KUKA KRL program: MyProgram_111().src

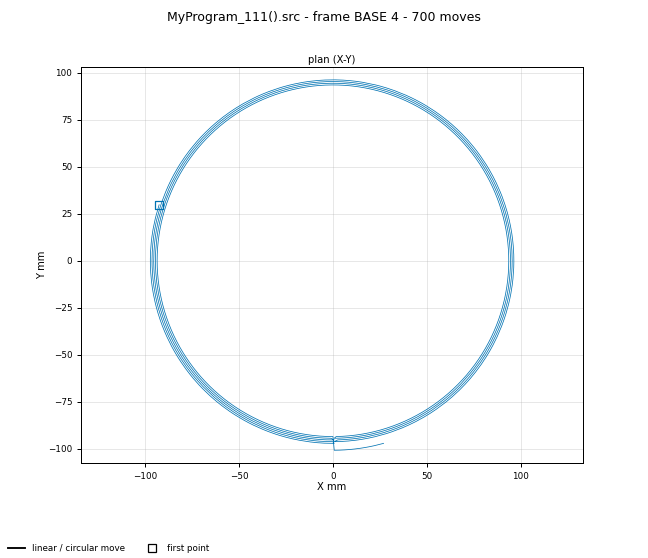
[picture p0: tool path of MyProgram_111().src in frame BASE 4, 700 of 700 moves have a stored position in this frame; points joined in program order, loops and branches not executed]
&ACCESS RVP
&REL 1
&PARAM TEMPLATE = C:\KRC\Roboter\Template\vorgabe
&PARAM EDITMASK = *
DEF MyProgram_111()
; ---- Setting reference (Base) ----
$BASE = BASE_DATA[4]

; --------------------------
; ---- Setting tool (TCP) ----
$TOOL = TOOL_DATA[3]
; --------------------------

$VEL.CP = VEL_APROX_PRINT
Startdeposition()
$VEL.CP = VEL_PRINT
LIN {X -92.4915,Y 29.7946,Z 97,A 157.868,B 24.9225,C -2.0326,E1 24.8471,E2 287.401} C_DIS
LIN {X -94.4382,Y 22.8874,Z 97,A 162.0208,B 24.9237,C -2.0166,E1 24.844,E2 283.2622} C_DIS
LIN {X -95.7031,Y 16.8359,Z 97,A 165.9283,B 24.924,C -2.0135,E1 24.8419,E2 279.3391} C_DIS
LIN {X -96.2599,Y 13.2878,Z 97,A 167.8285,B 24.925,C -1.9996,E1 24.8411,E2 277.4607} C_DIS
LIN {X -96.6738,Y 9.8311,Z 97,A 170.0082,B 24.9252,C -1.9971,E1 24.8405,E2 275.2738} C_DIS
LIN {X -97.0459,Y 4.9634,Z 97,A 172.6353,B 24.9265,C -1.9797,E1 24.84,E2 272.6726} C_DIS
LIN {X -97.1667,Y 1.1606,Z 97,A 174.9618,B 24.9269,C -1.9751,E1 24.8398,E2 270.3429} C_DIS
LIN {X -97.1555,Y -1.7889,Z 97,A 176.8668,B 24.9269,C -1.975,E1 24.8398,E2 268.4268} C_DIS
LIN {X -96.9581,Y -6.4444,Z 97,A 179.9808,B 24.9266,C -1.9782,E1 24.8403,E2 265.2864} C_DIS
LIN {X -96.5322,Y -11.1337,Z 97,A -177.5959,B 24.9281,C -1.9578,E1 24.841,E2 262.8972} C_DIS
LIN {X -96.1039,Y -14.3757,Z 97,A -175.1891,B 24.9274,C -1.9674,E1 24.842,E2 260.4532} C_DIS
LIN {X -95.5709,Y -17.5708,Z 97,A -174.0896,B 24.9298,C -1.9349,E1 24.8425,E2 259.4247} C_DIS
LIN {X -94.6671,Y -21.921,Z 97,A -171.138,B 24.9296,C -1.9376,E1 24.8442,E2 256.4493} C_DIS
LIN {X -94.0208,Y -24.5484,Z 97,A -168.9937,B 24.9287,C -1.9508,E1 24.8458,E2 254.261} C_DIS
LIN {X -93.1291,Y -27.7365,Z 97,A -167.1259,B 24.9293,C -1.9421,E1 24.8472,E2 252.4031} C_DIS
LIN {X -91.8935,Y -31.5962,Z 97,A -165.2192,B 24.931,C -1.919,E1 24.8489,E2 250.5406} C_DIS
LIN {X -90.915,Y -34.3054,Z 97,A -163.416,B 24.931,C -1.9175,E1 24.8506,E2 248.7308} C_DIS
LIN {X -89.6794,Y -37.418,Z 97,A -161.4125,B 24.9314,C -1.9127,E1 24.8527,E2 246.7275} C_DIS
LIN {X -88.3292,Y -40.505,Z 97,A -158.9881,B 24.9308,C -1.9216,E1 24.8556,E2 244.2687} C_DIS
LIN {X -85.934,Y -45.3624,Z 97,A -155.9633,B 24.9318,C -1.9072,E1 24.8594,E2 241.262} C_DIS
LIN {X -84.4252,Y -48.1133,Z 97,A -154.2857,B 24.9326,C -1.8964,E1 24.8617,E2 239.6013} C_DIS
LIN {X -82.6777,Y -51.0591,Z 97,A -152.4701,B 24.9334,C -1.8843,E1 24.8642,E2 237.8053} C_DIS
LIN {X -81.1737,Y -53.4156,Z 97,A -150.6577,B 24.9334,C -1.8856,E1 24.867,E2 235.9808} C_DIS
LIN {X -78.2895,Y -57.5602,Z 97,A -147.9461,B 24.9345,C -1.8692,E1 24.8714,E2 233.2948} C_DIS
LIN {X -76.0614,Y -60.4742,Z 97,A -145.6413,B 24.9345,C -1.8687,E1 24.8753,E2 230.9802} C_DIS
LIN {X -74.3345,Y -62.5867,Z 97,A -143.0069,B 24.9323,C -1.8998,E1 24.8802,E2 228.2597} C_DIS
LIN {X -71.1942,Y -66.1371,Z 97,A -141.1694,B 24.9351,C -1.8609,E1 24.8835,E2 226.5067} C_DIS
LIN {X -69.3992,Y -68.0168,Z 97,A -138.452,B 24.9325,C -1.8982,E1 24.889,E2 223.6888} C_DIS
LIN {X -65.4486,Y -71.8261,Z 97,A -136.4982,B 24.936,C -1.8476,E1 24.8928,E2 221.8475} C_DIS
LIN {X -61.836,Y -74.9588,Z 97,A -133.6287,B 24.9363,C -1.8439,E1 24.8989,E2 218.9758} C_DIS
LIN {X -59.0106,Y -77.2029,Z 97,A -131.1944,B 24.9358,C -1.8506,E1 24.9043,E2 216.5166} C_DIS
LIN {X -55.0989,Y -80.0414,Z 97,A -127.9514,B 24.9352,C -1.8594,E1 24.9117,E2 213.2414} C_DIS
LIN {X -52.3049,Y -81.8941,Z 97,A -126.3944,B 24.9364,C -1.8418,E1 24.9153,E2 211.7214} C_DIS
LIN {X -47.6565,Y -84.6838,Z 97,A -123.5051,B 24.9375,C -1.8265,E1 24.9222,E2 208.8597} C_DIS
LIN {X -44.9402,Y -86.1564,Z 97,A -121.5459,B 24.9373,C -1.8289,E1 24.927,E2 206.8894} C_DIS
LIN {X -42.2462,Y -87.5082,Z 97,A -119.4558,B 24.9367,C -1.8377,E1 24.9323,E2 204.7729} C_DIS
LIN {X -37.2841,Y -89.7359,Z 97,A -116.4957,B 24.9375,C -1.8255,E1 24.9399,E2 201.8348} C_DIS
LIN {X -34.0837,Y -90.9986,Z 97,A -114.3639,B 24.9375,C -1.8272,E1 24.9454,E2 199.6942} C_DIS
LIN {X -30.4442,Y -92.2814,Z 97,A -112.2394,B 24.9379,C -1.82,E1 24.951,E2 197.583} C_DIS
LIN {X -28.0314,Y -93.0419,Z 97,A -110.5722,B 24.9376,C -1.8251,E1 24.9555,E2 195.9006} C_DIS
LIN {X -24.7478,Y -93.9695,Z 97,A -108.1059,B 24.9365,C -1.8402,E1 24.9623,E2 193.3949} C_DIS
LIN {X -21.4833,Y -94.7682,Z 97,A -106.8785,B 24.9384,C -1.8121,E1 24.9654,E2 192.2324} C_DIS
LIN {X -17.7571,Y -95.5374,Z 97,A -104.2589,B 24.9376,C -1.8247,E1 24.9727,E2 189.58} C_DIS
LIN {X -12.0154,Y -96.4274,Z 97,A -100.8841,B 24.9378,C -1.822,E1 24.982,E2 186.2087} C_DIS
LIN {X -8.4428,Y -96.8057,Z 97,A -98.2149,B 24.9364,C -1.842,E1 24.9896,E2 183.4909} C_DIS
LIN {X -4.6237,Y -97.0629,Z 97,A -96.7543,B 24.9384,C -1.813,E1 24.9935,E2 182.0985} C_DIS
LIN {X 0.694,Y -97.1695,Z 97,A -93.9172,B 24.9391,C -1.8027,E1 25.0013,E2 179.2858} C_DIS
Enddeposition()
LIN {X 0.694,Y -97.1695,Z 97,A -93.9172,B 24.9391,C -1.8027,E1 25.0013,E2 179.2858} C_DIS
Startdeposition()
$VEL.CP = VEL_PRINT
LIN {X -0.1063,Y -96.2686,Z 97,A -95.3472,B 24.9403,C -1.7844,E1 24.9972,E2 180.7591} C_DIS
LIN {X -3.6596,Y -96.1991,Z 97,A -96.7459,B 24.9386,C -1.8095,E1 24.9935,E2 182.0986} C_DIS
LIN {X -7.1701,Y -96.0013,Z 97,A -99.0523,B 24.9391,C -1.8018,E1 24.987,E2 184.4239} C_DIS
LIN {X -10.3776,Y -95.7072,Z 97,A -101.037,B 24.9393,C -1.7996,E1 24.9814,E2 186.4149} C_DIS
LIN {X -16.5386,Y -94.8376,Z 97,A -104.7525,B 24.9393,C -1.8001,E1 24.9712,E2 190.1325} C_DIS
LIN {X -20.308,Y -94.1013,Z 97,A -106.7067,B 24.9384,C -1.8127,E1 24.9659,E2 192.0591} C_DIS
LIN {X -22.8168,Y -93.5244,Z 97,A -108.7921,B 24.9397,C -1.7943,E1 24.9601,E2 194.1911} C_DIS
LIN {X -27.203,Y -92.3442,Z 97,A -111.1051,B 24.9386,C -1.8095,E1 24.954,E2 196.4716} C_DIS
LIN {X -30.6307,Y -91.2645,Z 97,A -113.1926,B 24.9384,C -1.8129,E1 24.9484,E2 198.5547} C_DIS
LIN {X -33.6837,Y -90.1833,Z 97,A -115.2946,B 24.9387,C -1.8086,E1 24.9429,E2 200.6712} C_DIS
LIN {X -36.8901,Y -88.9204,Z 97,A -117.1546,B 24.9381,C -1.8172,E1 24.9381,E2 202.5149} C_DIS
LIN {X -42.0764,Y -86.5863,Z 97,A -120.7767,B 24.9384,C -1.8129,E1 24.9289,E2 206.1561} C_DIS
LIN {X -44.7962,Y -85.2099,Z 97,A -122.6012,B 24.9383,C -1.8149,E1 24.9243,E2 207.9809} C_DIS
LIN {X -47.0298,Y -83.9978,Z 97,A -124.2047,B 24.9383,C -1.8139,E1 24.9204,E2 209.5914} C_DIS
LIN {X -50.4531,Y -81.989,Z 97,A -126.5088,B 24.938,C -1.8192,E1 24.9149,E2 211.8897} C_DIS
LIN {X -52.931,Y -80.4098,Z 97,A -128.9407,B 24.9393,C -1.7993,E1 24.9091,E2 214.3772} C_DIS
LIN {X -56.6092,Y -77.8648,Z 97,A -130.8407,B 24.9373,C -1.829,E1 24.905,E2 216.213} C_DIS
LIN {X -58.4653,Y -76.4812,Z 97,A -132.5565,B 24.9379,C -1.8202,E1 24.9011,E2 217.9559} C_DIS
LIN {X -62.9436,Y -72.8408,Z 97,A -135.7325,B 24.9369,C -1.8353,E1 24.8943,E2 221.1083} C_DIS
LIN {X -69.1499,Y -66.9759,Z 97,A -140.5168,B 24.9355,C -1.8556,E1 24.8847,E2 225.8638} C_DIS
LIN {X -73.3934,Y -62.2966,Z 97,A -144.6286,B 24.9357,C -1.8524,E1 24.877,E2 230.0016} C_DIS
LIN {X -75.3487,Y -59.9173,Z 97,A -146.6761,B 24.9359,C -1.8498,E1 24.8734,E2 232.0651} C_DIS
LIN {X -77.8768,Y -56.5928,Z 97,A -149.3083,B 24.9358,C -1.8511,E1 24.869,E2 234.7068} C_DIS
LIN {X -80.6335,Y -52.5917,Z 97,A -151.6927,B 24.9341,C -1.8749,E1 24.8654,E2 237.0464} C_DIS
LIN {X -81.8943,Y -50.6061,Z 97,A -153.2387,B 24.9341,C -1.8738,E1 24.8631,E2 238.6028} C_DIS
LIN {X -83.5244,Y -47.8655,Z 97,A -155.0065,B 24.9335,C -1.8831,E1 24.8606,E2 240.3577} C_DIS
LIN {X -85.7783,Y -43.6981,Z 97,A -157.9857,B 24.9333,C -1.8857,E1 24.8567,E2 243.3466} C_DIS
LIN {X -87.5768,Y -39.9744,Z 97,A -160.4617,B 24.9329,C -1.8921,E1 24.8537,E2 245.8207} C_DIS
LIN {X -88.8678,Y -37.0149,Z 97,A -162.449,B 24.9326,C -1.8955,E1 24.8516,E2 247.8109} C_DIS
LIN {X -90.1653,Y -33.7313,Z 97,A -164.534,B 24.9322,C -1.9022,E1 24.8495,E2 249.8917} C_DIS
LIN {X -91.1712,Y -30.9074,Z 97,A -167.3212,B 24.934,C -1.8758,E1 24.847,E2 252.7577} C_DIS
LIN {X -92.7753,Y -25.7,Z 97,A -169.5931,B 24.9312,C -1.9162,E1 24.8453,E2 254.9465} C_DIS
LIN {X -93.6014,Y -22.5015,Z 97,A -172.0952,B 24.9319,C -1.9053,E1 24.8436,E2 257.4892} C_DIS
LIN {X -94.3933,Y -18.9045,Z 97,A -173.5687,B 24.9298,C -1.9348,E1 24.8428,E2 258.9009} C_DIS
LIN {X -95.3216,Y -13.462,Z 97,A -176.997,B 24.9294,C -1.9405,E1 24.8412,E2 262.3358} C_DIS
LIN {X -95.7625,Y -9.8494,Z 97,A -179.7199,B 24.9302,C -1.9299,E1 24.8404,E2 265.1006} C_DIS
LIN {X -96.0521,Y -6.4361,Z 97,A 178.1629,B 24.9299,C -1.9339,E1 24.84,E2 267.2209} C_DIS
LIN {X -96.2279,Y -2.7676,Z 97,A 176.4444,B 24.9283,C -1.9556,E1 24.8398,E2 268.898} C_DIS
LIN {X -96.2681,Y 0.3084,Z 97,A 173.9579,B 24.9294,C -1.9409,E1 24.8398,E2 271.4346} C_DIS
LIN {X -96.1614,Y 4.5356,Z 97,A 172.4406,B 24.9265,C -1.9804,E1 24.84,E2 272.8668} C_DIS
LIN {X -95.8516,Y 8.9387,Z 97,A 169.4889,B 24.9266,C -1.9785,E1 24.8406,E2 275.8406} C_DIS
LIN {X -95.4419,Y 12.5827,Z 97,A 167.4434,B 24.9258,C -1.9899,E1 24.8413,E2 277.8713} C_DIS
LIN {X -94.8189,Y 16.6424,Z 97,A 164.3977,B 24.9266,C -1.9788,E1 24.8427,E2 280.9615} C_DIS
LIN {X -94.2033,Y 19.8342,Z 97,A 162.8144,B 24.9253,C -1.996,E1 24.8436,E2 282.5132} C_DIS
LIN {X -93.6552,Y 22.2809,Z 97,A 160.0692,B 24.9279,C -1.9616,E1 24.8455,E2 285.3564} C_DIS
LIN {X -91.9819,Y 28.4036,Z 97,A 157.5986,B 24.9239,C -2.0142,E1 24.8473,E2 287.7158} C_DIS
LIN {X -90.9839,Y 31.4572,Z 97,A 154.5779,B 24.9261,C -1.9854,E1 24.8502,E2 290.8223} C_DIS
LIN {X -89.0472,Y 36.5773,Z 97,A 151.982,B 24.9238,C -2.0161,E1 24.8528,E2 293.3597} C_DIS
LIN {X -87.6404,Y 39.8331,Z 97,A 149.8079,B 24.9235,C -2.0204,E1 24.8553,E2 295.5354} C_DIS
LIN {X -86.2622,Y 42.7349,Z 97,A 147.841,B 24.9232,C -2.0243,E1 24.8578,E2 297.5034} C_DIS
LIN {X -84.6982,Y 45.7566,Z 97,A 146.652,B 24.9207,C -2.0568,E1 24.8592,E2 298.6213} C_DIS
LIN {X -82.7301,Y 49.2264,Z 97,A 144.0967,B 24.9206,C -2.0578,E1 24.8628,E2 301.1876} C_DIS
LIN {X -81.391,Y 51.41,Z 97,A 142.0984,B 24.9214,C -2.047,E1 24.8658,E2 303.2218} C_DIS
LIN {X -78.721,Y 55.4119,Z 97,A 139.1346,B 24.9211,C -2.0517,E1 24.8705,E2 306.1889} C_DIS
LIN {X -76.305,Y 58.6939,Z 97,A 136.7507,B 24.9205,C -2.0596,E1 24.8745,E2 308.5656} C_DIS
LIN {X -72.7774,Y 63.0162,Z 97,A 133.1858,B 24.9204,C -2.0604,E1 24.8809,E2 312.145} C_DIS
LIN {X -70.4253,Y 65.6345,Z 97,A 131.55,B 24.9188,C -2.0803,E1 24.884,E2 313.7405} C_DIS
LIN {X -67.6647,Y 68.4757,Z 97,A 128.6745,B 24.9197,C -2.0694,E1 24.8897,E2 316.6542} C_DIS
LIN {X -65.0275,Y 70.9849,Z 97,A 126.5163,B 24.9193,C -2.0746,E1 24.8941,E2 318.8085} C_DIS
LIN {X -62.3518,Y 73.3464,Z 97,A 124.8919,B 24.9176,C -2.0955,E1 24.8975,E2 320.3895} C_DIS
LIN {X -58.4338,Y 76.5045,Z 97,A 121.6806,B 24.9176,C -2.0949,E1 24.9046,E2 323.6142} C_DIS
LIN {X -54.9913,Y 79.0151,Z 97,A 119.1069,B 24.9174,C -2.0988,E1 24.9104,E2 326.1874} C_DIS
LIN {X -51.533,Y 81.3147,Z 97,A 116.1285,B 24.9183,C -2.087,E1 24.9175,E2 329.2035} C_DIS
LIN {X -47.8726,Y 83.5204,Z 97,A 113.9285,B 24.9171,C -2.1027,E1 24.9228,E2 331.3726} C_DIS
LIN {X -41.8924,Y 86.6747,Z 97,A 110.3041,B 24.9155,C -2.1225,E1 24.9317,E2 334.9598} C_DIS
LIN {X -39.8287,Y 87.6424,Z 97,A 108.8219,B 24.9157,C -2.1204,E1 24.9355,E2 336.4507} C_DIS
LIN {X -37.2678,Y 88.7612,Z 97,A 107.175,B 24.9154,C -2.1233,E1 24.9397,E2 338.0944} C_DIS
LIN {X -33.9421,Y 90.0855,Z 97,A 105.1375,B 24.915,C -2.1293,E1 24.945,E2 340.1221} C_DIS
LIN {X -28.5804,Y 91.9271,Z 97,A 102.0567,B 24.9139,C -2.1432,E1 24.9531,E2 343.1756} C_DIS
LIN {X -26.6002,Y 92.5198,Z 97,A 99.971,B 24.916,C -2.1158,E1 24.9588,E2 345.3298} C_DIS
LIN {X -23.1497,Y 93.4432,Z 97,A 98.3572,B 24.9145,C -2.135,E1 24.9631,E2 346.9002} C_DIS
LIN {X -20.474,Y 94.0651,Z 97,A 96.4503,B 24.9151,C -2.1273,E1 24.9683,E2 348.8278} C_DIS
LIN {X -15.9853,Y 94.9311,Z 97,A 94.0207,B 24.9142,C -2.1393,E1 24.9749,E2 351.2315} C_DIS
LIN {X -12.802,Y 95.4134,Z 97,A 92.0226,B 24.9142,C -2.1377,E1 24.9805,E2 353.235} C_DIS
LIN {X -7.6508,Y 95.963,Z 97,A 89.0303,B 24.9139,C -2.1424,E1 24.9888,E2 356.2177} C_DIS
LIN {X -4.163,Y 96.1774,Z 97,A 86.9285,B 24.9139,C -2.1424,E1 24.9946,E2 358.3201} C_DIS
LIN {X 1.1849,Y 96.262,Z 97,A 83.4209,B 24.9148,C -2.1319,E1 25.0045,E2 361.8527} C_DIS
LIN {X 5.3529,Y 96.1185,Z 97,A 81.2928,B 24.9138,C -2.1443,E1 25.0103,E2 363.9506} C_DIS
LIN {X 8.6175,Y 95.8813,Z 97,A 79.3012,B 24.9138,C -2.1426,E1 25.0159,E2 365.9451} C_DIS
LIN {X 12.1982,Y 95.4917,Z 97,A 77.1548,B 24.9139,C -2.1422,E1 25.0218,E2 368.091} C_DIS
LIN {X 15.6937,Y 94.9798,Z 97,A 74.8864,B 24.9145,C -2.1357,E1 25.0281,E2 370.3725} C_DIS
LIN {X 22.781,Y 93.5332,Z 97,A 70.7418,B 24.9142,C -2.1393,E1 25.0394,E2 374.5033} C_DIS
LIN {X 25.0573,Y 92.9492,Z 97,A 69.1352,B 24.9148,C -2.1311,E1 25.0438,E2 376.1269} C_DIS
LIN {X 28.7594,Y 91.8716,Z 97,A 66.8778,B 24.9148,C -2.1307,E1 25.0498,E2 378.3813} C_DIS
LIN {X 32.8246,Y 90.4986,Z 97,A 64.5081,B 24.9145,C -2.135,E1 25.056,E2 380.736} C_DIS
LIN {X 38.8687,Y 88.0729,Z 97,A 60.6771,B 24.9147,C -2.1326,E1 25.0659,E2 384.5638} C_DIS
LIN {X 41.7242,Y 86.7555,Z 97,A 58.6642,B 24.9153,C -2.1253,E1 25.071,E2 386.5889} C_DIS
LIN {X 44.0379,Y 85.6046,Z 97,A 56.6873,B 24.9167,C -2.1074,E1 25.076,E2 388.6025} C_DIS
LIN {X 47.3152,Y 83.8385,Z 97,A 54.9623,B 24.9155,C -2.1221,E1 25.0801,E2 390.2878} C_DIS
LIN {X 49.6095,Y 82.5017,Z 97,A 52.5123,B 24.9182,C -2.0883,E1 25.0862,E2 392.8101} C_DIS
LIN {X 53.8888,Y 79.7711,Z 97,A 50.4443,B 24.9159,C -2.118,E1 25.0908,E2 394.801} C_DIS
LIN {X 56.8975,Y 77.6537,Z 97,A 48.1904,B 24.9164,C -2.1119,E1 25.0959,E2 397.0615} C_DIS
LIN {X 59.7862,Y 75.4523,Z 97,A 46.0467,B 24.9166,C -2.1086,E1 25.1006,E2 399.205} C_DIS
LIN {X 63.1591,Y 72.6526,Z 97,A 42.8742,B 24.9186,C -2.0829,E1 25.1075,E2 402.4259} C_DIS
LIN {X 66.1256,Y 69.9635,Z 97,A 41.057,B 24.9174,C -2.0988,E1 25.1111,E2 404.198} C_DIS
LIN {X 68.6689,Y 67.4691,Z 97,A 38.8708,B 24.9179,C -2.0918,E1 25.1154,E2 406.3914} C_DIS
LIN {X 71.4686,Y 64.4966,Z 97,A 36.5932,B 24.9179,C -2.0921,E1 25.1197,E2 408.6584} C_DIS
LIN {X 73.095,Y 62.6468,Z 97,A 35.2236,B 24.9179,C -2.0924,E1 25.1222,E2 410.0212} C_DIS
LIN {X 75.1292,Y 60.1941,Z 97,A 33.3527,B 24.9182,C -2.0888,E1 25.1255,E2 411.8918} C_DIS
LIN {X 76.6102,Y 58.2967,Z 97,A 31.8354,B 24.9187,C -2.0822,E1 25.1281,E2 413.4176} C_DIS
LIN {X 78.5024,Y 55.7212,Z 97,A 30.0024,B 24.9189,C -2.0801,E1 25.1311,E2 415.2468} C_DIS
LIN {X 81.6082,Y 51.0639,Z 97,A 26.652,B 24.9196,C -2.0708,E1 25.1362,E2 418.6024} C_DIS
LIN {X 83.1374,Y 48.5373,Z 97,A 24.1439,B 24.9221,C -2.0378,E1 25.1399,E2 421.1753} C_DIS
LIN {X 85.2358,Y 44.7471,Z 97,A 22.2783,B 24.9206,C -2.0576,E1 25.1422,E2 422.9844} C_DIS
LIN {X 86.8297,Y 41.5699,Z 97,A 20.4727,B 24.9202,C -2.0635,E1 25.1444,E2 424.7665} C_DIS
LIN {X 89.0364,Y 36.6069,Z 97,A 17.0287,B 24.9215,C -2.0461,E1 25.1483,E2 428.2326} C_DIS
LIN {X 89.9521,Y 34.2941,Z 97,A 14.7796,B 24.924,C -2.0127,E1 25.1506,E2 430.5481} C_DIS
LIN {X 91.4513,Y 30.0714,Z 97,A 12.1056,B 24.9247,C -2.0044,E1 25.1529,E2 433.2265} C_DIS
LIN {X 92.7719,Y 25.712,Z 97,A 10.1116,B 24.9232,C -2.0234,E1 25.1544,E2 435.1643} C_DIS
LIN {X 93.8162,Y 21.5858,Z 97,A 7.6077,B 24.9237,C -2.0167,E1 25.1561,E2 437.6694} C_DIS
LIN {X 94.5734,Y 17.9821,Z 97,A 5.4465,B 24.9242,C -2.0111,E1 25.1573,E2 439.8314} C_DIS
LIN {X 95.1599,Y 14.5614,Z 97,A 3.4483,B 24.9245,C -2.0072,E1 25.1581,E2 441.827} C_DIS
LIN {X 95.6181,Y 11.1625,Z 97,A 1.4693,B 24.9248,C -2.0031,E1 25.1588,E2 443.8039} C_DIS
LIN {X 95.947,Y 7.8507,Z 97,A -0.5562,B 24.9254,C -1.9951,E1 25.1594,E2 445.8364} C_DIS
LIN {X 96.2103,Y 3.3404,Z 97,A -3.7404,B 24.9274,C -1.9675,E1 25.1598,E2 449.0668} C_DIS
LIN {X 96.2683,Y -0.2759,Z 97,A -5.409,B 24.9266,C -1.9791,E1 25.1598,E2 450.698} C_DIS
LIN {X 96.1914,Y -3.8381,Z 97,A -7.1655,B 24.926,C -1.9863,E1 25.1596,E2 452.427} C_DIS
LIN {X 95.7875,Y -9.6102,Z 97,A -10.892,B 24.9277,C -1.9643,E1 25.1589,E2 456.1835} C_DIS
LIN {X 95.3861,Y -13.0079,Z 97,A -12.9595,B 24.9282,C -1.9565,E1 25.1581,E2 458.2571} C_DIS
LIN {X 94.6398,Y -17.6367,Z 97,A -15.7128,B 24.9288,C -1.949,E1 25.1568,E2 461.012} C_DIS
LIN {X 94.1134,Y -20.2525,Z 97,A -17.2967,B 24.9291,C -1.9441,E1 25.1559,E2 462.5982} C_DIS
LIN {X 93.4103,Y -23.2847,Z 97,A -19.3832,B 24.9302,C -1.9292,E1 25.1545,E2 464.7078} C_DIS
LIN {X 92.0627,Y -28.143,Z 97,A -22.0736,B 24.93,C -1.9317,E1 25.1524,E2 467.377} C_DIS
LIN {X 91.0382,Y -31.3019,Z 97,A -24.0007,B 24.9304,C -1.9274,E1 25.1507,E2 469.3033} C_DIS
LIN {X 89.7528,Y -34.8143,Z 97,A -26.5939,B 24.9319,C -1.9064,E1 25.1481,E2 471.9314} C_DIS
LIN {X 87.3524,Y -40.4601,Z 97,A -29.9301,B 24.9318,C -1.9074,E1 25.1444,E2 475.247} C_DIS
LIN {X 85.121,Y -44.965,Z 97,A -33.3271,B 24.9335,C -1.8831,E1 25.14,E2 478.6835} C_DIS
LIN {X 83.4643,Y -47.9701,Z 97,A -34.9806,B 24.9329,C -1.892,E1 25.1378,E2 480.3074} C_DIS
LIN {X 81.504,Y -51.2308,Z 97,A -36.8015,B 24.9321,C -1.9025,E1 25.1352,E2 482.0942} C_DIS
LIN {X 78.9338,Y -55.1082,Z 97,A -39.7281,B 24.9331,C -1.8887,E1 25.1306,E2 485.039} C_DIS
LIN {X 75.772,Y -59.3818,Z 97,A -43.0489,B 24.9342,C -1.8741,E1 25.125,E2 488.3783} C_DIS
LIN {X 73.0117,Y -62.7429,Z 97,A -45.7233,B 24.9349,C -1.8641,E1 25.1202,E2 491.0641} C_DIS
LIN {X 70.3161,Y -65.7502,Z 97,A -48.2366,B 24.9356,C -1.8539,E1 25.1154,E2 493.5904} C_DIS
LIN {X 67.3056,Y -68.8304,Z 97,A -50.4053,B 24.935,C -1.8625,E1 25.1112,E2 495.7294} C_DIS
LIN {X 63.5474,Y -72.3135,Z 97,A -53.6784,B 24.9361,C -1.847,E1 25.1044,E2 499.0262} C_DIS
LIN {X 60.019,Y -75.2683,Z 97,A -56.3101,B 24.9361,C -1.8449,E1 25.0988,E2 501.6527} C_DIS
LIN {X 54.9405,Y -79.0504,Z 97,A -60.6156,B 24.9381,C -1.8171,E1 25.0889,E2 506.0087} C_DIS
LIN {X 51.8209,Y -81.1299,Z 97,A -62.3338,B 24.9371,C -1.8318,E1 25.085,E2 507.6865} C_DIS
LIN {X 48.3856,Y -83.2256,Z 97,A -65.0835,B 24.9383,C -1.8143,E1 25.0783,E2 510.4693} C_DIS
LIN {X 43.9793,Y -85.6346,Z 97,A -67.6777,B 24.9377,C -1.8238,E1 25.072,E2 513.0337} C_DIS
LIN {X 40.7775,Y -87.2047,Z 97,A -69.7184,B 24.9377,C -1.8234,E1 25.0668,E2 515.07} C_DIS
LIN {X 36.9747,Y -88.8847,Z 97,A -72.4202,B 24.9385,C -1.8113,E1 25.0598,E2 517.7938} C_DIS
LIN {X 31.3237,Y -91.0307,Z 97,A -75.8848,B 24.9385,C -1.8114,E1 25.0508,E2 521.2509} C_DIS
LIN {X 28.2543,Y -92.0282,Z 97,A -78.1261,B 24.9394,C -1.7975,E1 25.0447,E2 523.5211} C_DIS
LIN {X 22.3363,Y -93.6415,Z 97,A -81.4234,B 24.9388,C -1.8066,E1 25.0359,E2 526.7919} C_DIS
LIN {X 19.14,Y -94.3458,Z 97,A -83.3011,B 24.9388,C -1.8074,E1 25.0308,E2 528.6652} C_DIS
LIN {X 15.3613,Y -95.0354,Z 97,A -85.5765,B 24.9388,C -1.806,E1 25.0245,E2 530.9416} C_DIS
LIN {X 12.2874,Y -95.4801,Z 97,A -87.3723,B 24.9388,C -1.8067,E1 25.0195,E2 532.7342} C_DIS
LIN {X 8.1215,Y -95.9254,Z 97,A -90.1215,B 24.9395,C -1.7961,E1 25.0118,E2 535.5067} C_DIS
LIN {X 3.9667,Y -96.1859,Z 97,A -92.4071,B 24.9391,C -1.802,E1 25.0055,E2 537.7774} C_DIS
LIN {X 0.6816,Y -96.2642,Z 97,A -93.5463,B 24.9372,C -1.8308,E1 25.0025,E2 538.8484} C_DIS
Enddeposition()
LIN {X 0.6816,Y -96.2642,Z 97,A -93.5463,B 24.9372,C -1.8308,E1 25.0025,E2 538.8484} C_DIS
Startdeposition()
$VEL.CP = VEL_PRINT
LIN {X 2.61,Y -95.3278,Z 97,A -92.3092,B 24.9359,C -1.8495,E1 25.0061,E2 537.567} C_DIS
LIN {X 5.9173,Y -95.1806,Z 97,A -89.9957,B 24.935,C -1.862,E1 25.0126,E2 535.2247} C_DIS
LIN {X 10.4074,Y -94.7946,Z 97,A -87.787,B 24.9362,C -1.8454,E1 25.0187,E2 533.0567} C_DIS
LIN {X 12.8089,Y -94.5005,Z 97,A -86.1366,B 24.9356,C -1.8535,E1 25.0233,E2 531.3886} C_DIS
LIN {X 15.9028,Y -94.0278,Z 97,A -84.2836,B 24.9356,C -1.8539,E1 25.0284,E2 529.5364} C_DIS
LIN {X 19.0921,Y -93.4323,Z 97,A -82.3681,B 24.9356,C -1.8543,E1 25.0336,E2 527.6222} C_DIS
LIN {X 24.8011,Y -92.0816,Z 97,A -78.9921,B 24.9356,C -1.8524,E1 25.0428,E2 524.2558} C_DIS
LIN {X 27.4548,Y -91.3261,Z 97,A -77.1848,B 24.9352,C -1.8597,E1 25.0476,E2 522.4342} C_DIS
LIN {X 30.8104,Y -90.2494,Z 97,A -75.0091,B 24.9348,C -1.8644,E1 25.0534,E2 520.2515} C_DIS
LIN {X 33.9489,Y -89.1157,Z 97,A -72.5761,B 24.9335,C -1.8831,E1 25.0599,E2 517.7796} C_DIS
LIN {X 37.1197,Y -87.8421,Z 97,A -70.8465,B 24.9342,C -1.874,E1 25.0643,E2 516.0755} C_DIS
LIN {X 40.7737,Y -86.2088,Z 97,A -68.1737,B 24.9332,C -1.8878,E1 25.0711,E2 513.377} C_DIS
LIN {X 44.9241,Y -84.1203,Z 97,A -65.8946,B 24.9342,C -1.8733,E1 25.0767,E2 511.1385} C_DIS
LIN {X 49.5049,Y -81.5069,Z 97,A -63.1252,B 24.9349,C -1.8641,E1 25.0833,E2 508.3991} C_DIS
LIN {X 52.7006,Y -79.4784,Z 97,A -60.1397,B 24.9327,C -1.8952,E1 25.0904,E2 505.3499} C_DIS
LIN {X 58.8479,Y -75.041,Z 97,A -56.098,B 24.9334,C -1.8852,E1 25.0994,E2 501.3461} C_DIS
LIN {X 61.5803,Y -72.8155,Z 97,A -53.6713,B 24.9322,C -1.9016,E1 25.1047,E2 498.8898} C_DIS
LIN {X 64.8543,Y -69.9145,Z 97,A -50.8739,B 24.9313,C -1.9142,E1 25.1105,E2 496.074} C_DIS
LIN {X 67.3983,Y -67.4675,Z 97,A -48.5764,B 24.9304,C -1.9261,E1 25.1151,E2 493.7581} C_DIS
LIN {X 69.6648,Y -65.1217,Z 97,A -46.9572,B 24.931,C -1.918,E1 25.1182,E2 492.1652} C_DIS
LIN {X 72.314,Y -62.1681,Z 97,A -44.6332,B 24.9308,C -1.9218,E1 25.1224,E2 489.8426} C_DIS
LIN {X 74.6924,Y -59.289,Z 97,A -42.8363,B 24.9316,C -1.9106,E1 25.1255,E2 488.0804} C_DIS
LIN {X 78.4391,Y -54.2353,Z 97,A -38.4662,B 24.9292,C -1.9435,E1 25.1328,E2 483.6537} C_DIS
LIN {X 80.659,Y -50.8763,Z 97,A -36.3307,B 24.9295,C -1.9394,E1 25.136,E2 481.5387} C_DIS
LIN {X 82.2957,Y -48.1838,Z 97,A -34.0702,B 24.928,C -1.9591,E1 25.1393,E2 479.2434} C_DIS
LIN {X 84.4591,Y -44.2809,Z 97,A -31.0116,B 24.9264,C -1.9817,E1 25.1433,E2 476.1475} C_DIS
LIN {X 86.4472,Y -40.2614,Z 97,A -29.5592,B 24.9293,C -1.9416,E1 25.145,E2 474.7975} C_DIS
LIN {X 87.7634,Y -37.3065,Z 97,A -26.7073,B 24.9263,C -1.9827,E1 25.1482,E2 471.8644} C_DIS
LIN {X 89.0408,Y -34.1466,Z 97,A -25.386,B 24.9279,C -1.9608,E1 25.1495,E2 470.6021} C_DIS
LIN {X 90.3278,Y -30.5779,Z 97,A -22.8768,B 24.9267,C -1.9767,E1 25.1518,E2 468.0693} C_DIS
LIN {X 91.4215,Y -27.1332,Z 97,A -20.7574,B 24.9264,C -1.9815,E1 25.1536,E2 465.9506} C_DIS
LIN {X 92.7543,Y -22.1573,Z 97,A -17.5724,B 24.9254,C -1.9948,E1 25.1558,E2 462.7527} C_DIS
LIN {X 93.4717,Y -18.9002,Z 97,A -15.5859,B 24.925,C -2.0005,E1 25.157,E2 460.7642} C_DIS
LIN {X 94.1569,Y -15.1295,Z 97,A -13.5227,B 24.9251,C -1.9986,E1 25.1579,E2 458.7176} C_DIS
LIN {X 94.524,Y -12.628,Z 97,A -11.8216,B 24.9242,C -2.0106,E1 25.1586,E2 456.9983} C_DIS
LIN {X 94.9298,Y -9.0849,Z 97,A -9.2181,B 24.9223,C -2.0354,E1 25.1593,E2 454.3516} C_DIS
LIN {X 95.2022,Y -5.5427,Z 97,A -7.9237,B 24.9243,C -2.0097,E1 25.1596,E2 453.1257} C_DIS
LIN {X 95.3146,Y -3.0397,Z 97,A -6.1842,B 24.9232,C -2.0236,E1 25.1597,E2 451.3637} C_DIS
LIN {X 95.3641,Y 0.2359,Z 97,A -3.8011,B 24.9215,C -2.046,E1 25.1597,E2 448.9419} C_DIS
LIN {X 95.2214,Y 5.1962,Z 97,A -1.4361,B 24.9226,C -2.0317,E1 25.1595,E2 446.6248} C_DIS
LIN {X 95.0468,Y 7.7612,Z 97,A 0.3877,B 24.9214,C -2.0474,E1 25.1591,E2 444.7747} C_DIS
LIN {X 94.6935,Y 11.282,Z 97,A 2.518,B 24.9209,C -2.0543,E1 25.1585,E2 442.6407} C_DIS
LIN {X 94.208,Y 14.7987,Z 97,A 4.6359,B 24.9204,C -2.0604,E1 25.1576,E2 440.5208} C_DIS
LIN {X 93.5954,Y 18.2774,Z 97,A 6.6408,B 24.9202,C -2.0625,E1 25.1566,E2 438.5227} C_DIS
LIN {X 92.1897,Y 24.4006,Z 97,A 10.4181,B 24.9193,C -2.0742,E1 25.1541,E2 434.7397} C_DIS
LIN {X 90.9973,Y 28.5251,Z 97,A 13.1802,B 24.9182,C -2.089,E1 25.1519,E2 431.9584} C_DIS
LIN {X 89.2622,Y 33.5621,Z 97,A 16.0474,B 24.9184,C -2.0857,E1 25.1492,E2 429.1152} C_DIS
LIN {X 88.2146,Y 36.2267,Z 97,A 17.7943,B 24.918,C -2.0917,E1 25.1474,E2 427.3637} C_DIS
LIN {X 86.3913,Y 40.3816,Z 97,A 20.4319,B 24.9176,C -2.0961,E1 25.1444,E2 424.7301} C_DIS
LIN {X 85.1371,Y 42.9652,Z 97,A 22.3249,B 24.9167,C -2.1072,E1 25.142,E2 422.8209} C_DIS
LIN {X 82.9912,Y 46.9746,Z 97,A 25.0888,B 24.916,C -2.1159,E1 25.1383,E2 420.051} C_DIS
LIN {X 81.084,Y 50.196,Z 97,A 27.2824,B 24.9157,C -2.1197,E1 25.1351,E2 417.8596} C_DIS
LIN {X 78.5077,Y 54.1365,Z 97,A 30.078,B 24.9153,C -2.1257,E1 25.1308,E2 415.0638} C_DIS
LIN {X 76.5977,Y 56.8087,Z 97,A 32.3455,B 24.914,C -2.1417,E1 25.127,E2 412.7694} C_DIS
LIN {X 72.4677,Y 61.9885,Z 97,A 35.5901,B 24.9154,C -2.1234,E1 25.1214,E2 409.583} C_DIS
LIN {X 70.99,Y 63.6752,Z 97,A 37.3079,B 24.9141,C -2.1403,E1 25.1182,E2 407.8329} C_DIS
LIN {X 67.4682,Y 67.3976,Z 97,A 40.2156,B 24.9141,C -2.1406,E1 25.1126,E2 404.9372} C_DIS
LIN {X 63.5594,Y 71.0936,Z 97,A 44.0568,B 24.9117,C -2.1699,E1 25.1046,E2 401.0422} C_DIS
LIN {X 61.0506,Y 73.2594,Z 97,A 45.5638,B 24.9128,C -2.1557,E1 25.1014,E2 399.5747} C_DIS
LIN {X 57.8449,Y 75.8174,Z 97,A 48.4771,B 24.9111,C -2.1768,E1 25.0949,E2 396.6222} C_DIS
LIN {X 54.4827,Y 78.2671,Z 97,A 50.5012,B 24.9122,C -2.1634,E1 25.0904,E2 394.6367} C_DIS
LIN {X 50.0687,Y 81.1635,Z 97,A 53.5285,B 24.9122,C -2.1631,E1 25.0833,E2 391.6201} C_DIS
LIN {X 46.9644,Y 82.9983,Z 97,A 55.9148,B 24.9113,C -2.1742,E1 25.0775,E2 389.2146} C_DIS
LIN {X 43.5469,Y 84.8398,Z 97,A 58.1543,B 24.9113,C -2.174,E1 25.072,E2 386.9821} C_DIS
LIN {X 40.4426,Y 86.3629,Z 97,A 59.9657,B 24.9119,C -2.1668,E1 25.0675,E2 385.1923} C_DIS
LIN {X 38.0367,Y 87.449,Z 97,A 62.2818,B 24.9096,C -2.1951,E1 25.0614,E2 382.815} C_DIS
LIN {X 34.9931,Y 88.7108,Z 97,A 63.6026,B 24.9114,C -2.1732,E1 25.0581,E2 381.5489} C_DIS
LIN {X 32.5285,Y 89.6439,Z 97,A 65.4661,B 24.9105,C -2.1848,E1 25.0532,E2 379.662} C_DIS
LIN {X 28.9136,Y 90.8753,Z 97,A 67.8042,B 24.9102,C -2.1882,E1 25.047,E2 377.3202} C_DIS
LIN {X 23.1403,Y 92.5145,Z 97,A 72.363,B 24.9071,C -2.2248,E1 25.0345,E2 372.6817} C_DIS
LIN {X 17.7268,Y 93.7014,Z 97,A 74.4838,B 24.9106,C -2.183,E1 25.0289,E2 370.6627} C_DIS
LIN {X 15.0426,Y 94.1703,Z 97,A 76.1567,B 24.9105,C -2.1848,E1 25.0243,E2 368.9872} C_DIS
LIN {X 12.1208,Y 94.5897,Z 97,A 78.0295,B 24.9101,C -2.1887,E1 25.0191,E2 367.1067} C_DIS
LIN {X 8.5712,Y 94.9772,Z 97,A 80.2193,B 24.91,C -2.1905,E1 25.013,E2 364.9139} C_DIS
LIN {X 5.0548,Y 95.2292,Z 97,A 82.3518,B 24.91,C -2.191,E1 25.0071,E2 362.7811} C_DIS
LIN {X 0.9928,Y 95.3587,Z 97,A 84.9324,B 24.9096,C -2.1956,E1 24.9998,E2 360.1901} C_DIS
LIN {X -3.326,Y 95.3058,Z 97,A 87.3071,B 24.9103,C -2.1872,E1 24.9933,E2 357.835} C_DIS
LIN {X -6.834,Y 95.1187,Z 97,A 89.5095,B 24.9101,C -2.1895,E1 24.9871,E2 355.6264} C_DIS
LIN {X -10.874,Y 94.7413,Z 97,A 91.8289,B 24.9105,C -2.1842,E1 24.9807,E2 353.3184} C_DIS
LIN {X -13.7644,Y 94.3651,Z 97,A 93.6967,B 24.9103,C -2.1871,E1 24.9755,E2 351.4422} C_DIS
LIN {X -17.2061,Y 93.7985,Z 97,A 96.3477,B 24.9088,C -2.2046,E1 24.9681,E2 348.7469} C_DIS
LIN {X -21.056,Y 93.0103,Z 97,A 97.9708,B 24.9111,C -2.1772,E1 24.9639,E2 347.1868} C_DIS
LIN {X -24.1344,Y 92.259,Z 97,A 100.5156,B 24.9094,C -2.1972,E1 24.9568,E2 344.5909} C_DIS
LIN {X -27.57,Y 91.2919,Z 97,A 102.2813,B 24.9107,C -2.1819,E1 24.9522,E2 342.8585} C_DIS
LIN {X -32.0736,Y 89.809,Z 97,A 104.8049,B 24.9119,C -2.1675,E1 24.9456,E2 340.3645} C_DIS
LIN {X -35.942,Y 88.3305,Z 97,A 107.5112,B 24.9116,C -2.1714,E1 24.9385,E2 337.6429} C_DIS
LIN {X -39.8295,Y 86.6483,Z 97,A 109.843,B 24.9124,C -2.1606,E1 24.9326,E2 335.3315} C_DIS
LIN {X -42.5819,Y 85.3285,Z 97,A 113.0742,B 24.9088,C -2.2046,E1 24.9243,E2 331.9869} C_DIS
LIN {X -47.7915,Y 82.5238,Z 97,A 115.1585,B 24.9134,C -2.1491,E1 24.9195,E2 330.0285} C_DIS
LIN {X -50.8871,Y 80.6523,Z 97,A 117.4605,B 24.9134,C -2.1493,E1 24.914,E2 327.7189} C_DIS
LIN {X -52.9329,Y 79.3251,Z 97,A 119.455,B 24.9122,C -2.164,E1 24.9093,E2 325.683} C_DIS
LIN {X -56.586,Y 76.7608,Z 97,A 122.6065,B 24.9113,C -2.1741,E1 24.9021,E2 322.4964} C_DIS
LIN {X -60.1509,Y 73.9999,Z 97,A 124.4033,B 24.9143,C -2.1381,E1 24.8983,E2 320.7784} C_DIS
LIN {X -62.506,Y 72.0221,Z 97,A 126.6433,B 24.9136,C -2.1468,E1 24.8935,E2 318.5091} C_DIS
LIN {X -66.1305,Y 68.7085,Z 97,A 129.7208,B 24.9138,C -2.144,E1 24.8872,E2 315.4255} C_DIS
LIN {X -69.5305,Y 65.2658,Z 97,A 132.2492,B 24.9153,C -2.1246,E1 24.8824,E2 312.9325} C_DIS
LIN {X -72.1107,Y 62.4046,Z 97,A 134.6536,B 24.9156,C -2.1216,E1 24.878,E2 310.5245} C_DIS
LIN {X -75.7447,Y 57.9392,Z 97,A 138.1477,B 24.9162,C -2.1136,E1 24.8719,E2 307.0331} C_DIS
LIN {X -78.9356,Y 53.5096,Z 97,A 142.3036,B 24.9147,C -2.133,E1 24.8652,E2 302.8103} C_DIS
LIN {X -81.6145,Y 49.3278,Z 97,A 144.1341,B 24.9183,C -2.0873,E1 24.8626,E2 301.0797} C_DIS
LIN {X -83.1873,Y 46.6261,Z 97,A 146.2054,B 24.9183,C -2.088,E1 24.8597,E2 298.9957} C_DIS
LIN {X -86.0957,Y 41.0091,Z 97,A 149.8811,B 24.9194,C -2.0728,E1 24.8551,E2 295.3368} C_DIS
LIN {X -87.1781,Y 38.6575,Z 97,A 151.7343,B 24.9191,C -2.0776,E1 24.8529,E2 293.462} C_DIS
LIN {X -90.1449,Y 31.1166,Z 97,A 156.36,B 24.9208,C -2.0548,E1 24.8483,E2 288.8647} C_DIS
LIN {X -91.2892,Y 27.5793,Z 97,A 159.5503,B 24.919,C -2.0784,E1 24.8457,E2 285.5995} C_DIS
LIN {X -92.422,Y 23.502,Z 97,A 161.3775,B 24.9214,C -2.0474,E1 24.8444,E2 283.8356} C_DIS
LIN {X -93.2191,Y 20.1084,Z 97,A 163.5525,B 24.9217,C -2.0434,E1 24.8431,E2 281.6576} C_DIS
LIN {X -93.9347,Y 16.4488,Z 97,A 166.3382,B 24.9209,C -2.0536,E1 24.8417,E2 278.8309} C_DIS
LIN {X -94.5132,Y 12.7111,Z 97,A 167.8295,B 24.9234,C -2.0214,E1 24.8411,E2 277.4076} C_DIS
LIN {X -94.8489,Y 9.8891,Z 97,A 170.6561,B 24.9211,C -2.0517,E1 24.8403,E2 274.4916} C_DIS
LIN {X -95.2319,Y 5.0049,Z 97,A 172.1116,B 24.9254,C -1.9948,E1 24.84,E2 273.1633} C_DIS
LIN {X -95.3619,Y -0.551,Z 97,A 175.9605,B 24.925,C -2.0001,E1 24.8398,E2 269.2786} C_DIS
LIN {X -95.2606,Y -4.4167,Z 97,A 178.5201,B 24.925,C -2.0001,E1 24.84,E2 266.7035} C_DIS
LIN {X -94.9934,Y -8.3889,Z 97,A -178.9943,B 24.9253,C -1.9955,E1 24.8406,E2 264.214} C_DIS
LIN {X -94.5703,Y -12.2705,Z 97,A -176.3483,B 24.9252,C -1.9977,E1 24.8415,E2 261.5468} C_DIS
LIN {X -94.0882,Y -15.542,Z 97,A -174.6941,B 24.9264,C -1.9808,E1 24.8422,E2 259.9232} C_DIS
LIN {X -93.6143,Y -18.1792,Z 97,A -172.5851,B 24.9256,C -1.9919,E1 24.8434,E2 257.7753} C_DIS
LIN {X -92.8022,Y -21.9571,Z 97,A -170.7985,B 24.9274,C -1.9674,E1 24.8445,E2 256.0366} C_DIS
LIN {X -91.9819,Y -25.1698,Z 97,A -168.8691,B 24.928,C -1.9594,E1 24.8459,E2 254.1152} C_DIS
LIN {X -90.4489,Y -30.2186,Z 97,A -165.6528,B 24.9286,C -1.9513,E1 24.8486,E2 250.8996} C_DIS
LIN {X -89.3548,Y -33.3175,Z 97,A -163.5859,B 24.9288,C -1.9485,E1 24.8505,E2 248.8277} C_DIS
LIN {X -88.0687,Y -36.582,Z 97,A -161.5009,B 24.9293,C -1.9416,E1 24.8527,E2 246.7475} C_DIS
LIN {X -86.8299,Y -39.4303,Z 97,A -159.3442,B 24.929,C -1.9458,E1 24.8552,E2 244.5691} C_DIS
LIN {X -84.99,Y -43.253,Z 97,A -156.6942,B 24.9293,C -1.942,E1 24.8585,E2 241.9138} C_DIS
LIN {X -83.1187,Y -46.7489,Z 97,A -154.7243,B 24.9307,C -1.9221,E1 24.8611,E2 239.9811} C_DIS
LIN {X -81.5002,Y -49.5159,Z 97,A -152.7937,B 24.9311,C -1.9171,E1 24.8639,E2 238.0523} C_DIS
LIN {X -79.9749,Y -51.9459,Z 97,A -150.9737,B 24.9311,C -1.9158,E1 24.8666,E2 236.2263} C_DIS
LIN {X -77.7472,Y -55.2225,Z 97,A -148.6847,B 24.9318,C -1.9068,E1 24.8703,E2 233.9473} C_DIS
LIN {X -75.9766,Y -57.6356,Z 97,A -146.6665,B 24.9316,C -1.9097,E1 24.8737,E2 231.9127} C_DIS
LIN {X -73.4563,Y -60.8137,Z 97,A -144.3939,B 24.9324,C -1.8985,E1 24.8776,E2 229.656} C_DIS
LIN {X -69.9449,Y -64.8232,Z 97,A -141.3641,B 24.9333,C -1.8856,E1 24.8832,E2 226.6435} C_DIS
LIN {X -67.0982,Y -67.7639,Z 97,A -137.9459,B 24.9314,C -1.9124,E1 24.8901,E2 223.1469} C_DIS
LIN {X -63.9266,Y -70.7649,Z 97,A -136.2783,B 24.9341,C -1.8751,E1 24.8934,E2 221.5615} C_DIS
LIN {X -60.6198,Y -73.6174,Z 97,A -133.5148,B 24.9341,C -1.8747,E1 24.8993,E2 218.7882} C_DIS
LIN {X -57.7178,Y -75.9148,Z 97,A -131.3402,B 24.9345,C -1.869,E1 24.904,E2 216.6191} C_DIS
LIN {X -53.3801,Y -79.0232,Z 97,A -128.0214,B 24.9346,C -1.8675,E1 24.9116,E2 213.2926} C_DIS
LIN {X -50.5651,Y -80.8534,Z 97,A -125.964,B 24.9347,C -1.8657,E1 24.9165,E2 211.2327} C_DIS
LIN {X -47.4083,Y -82.744,Z 97,A -123.8647,B 24.9352,C -1.8588,E1 24.9215,E2 209.1436} C_DIS
LIN {X -45.2571,Y -83.9402,Z 97,A -122.1467,B 24.9348,C -1.8649,E1 24.9258,E2 207.4061} C_DIS
LIN {X -42.7323,Y -85.2539,Z 97,A -120.4882,B 24.9351,C -1.861,E1 24.9299,E2 205.7525} C_DIS
LIN {X -38.1111,Y -87.4165,Z 97,A -117.4933,B 24.9355,C -1.8551,E1 24.9375,E2 202.7641} C_DIS
LIN {X -34.9939,Y -88.7105,Z 97,A -115.4341,B 24.9355,C -1.8542,E1 24.9428,E2 200.7027} C_DIS
LIN {X -31.9314,Y -89.8589,Z 97,A -113.3293,B 24.9353,C -1.8573,E1 24.9484,E2 198.5863} C_DIS
LIN {X -26.6217,Y -91.5732,Z 97,A -110.3049,B 24.9363,C -1.8434,E1 24.9564,E2 195.5895} C_DIS
LIN {X -20.991,Y -93.0254,Z 97,A -106.9292,B 24.9367,C -1.8372,E1 24.9655,E2 192.2236} C_DIS
LIN {X -17.3878,Y -93.7658,Z 97,A -104.3042,B 24.9358,C -1.8508,E1 24.9727,E2 189.5633} C_DIS
LIN {X -12.5998,Y -94.5276,Z 97,A -101.5746,B 24.9363,C -1.8437,E1 24.9802,E2 186.8484} C_DIS
LIN {X -9.7484,Y -94.8636,Z 97,A -99.7975,B 24.9362,C -1.8453,E1 24.9852,E2 185.0664} C_DIS
LIN {X -6.5384,Y -95.1387,Z 97,A -97.6512,B 24.9357,C -1.8528,E1 24.9912,E2 182.9015} C_DIS
LIN {X -3.559,Y -95.2981,Z 97,A -95.6954,B 24.9352,C -1.8588,E1 24.9967,E2 180.931} C_DIS
LIN {X 0.6813,Y -95.3593,Z 97,A -94.2912,B 24.938,C -1.8186,E1 25.0004,E2 179.6221} C_DIS
Enddeposition()
LIN {X 0.6813,Y -95.3593,Z 97,A -94.2912,B 24.938,C -1.8186,E1 25.0004,E2 179.6221} C_DIS
Startdeposition()
$VEL.CP = VEL_PRINT
LIN {X -1.1523,Y -94.4532,Z 97,A -95.6762,B 24.9376,C -1.8247,E1 24.9965,E2 180.9926} C_DIS
LIN {X -5.0663,Y -94.3227,Z 97,A -97.9508,B 24.9374,C -1.828,E1 24.9902,E2 183.2599} C_DIS
LIN {X -8.4852,Y -94.0768,Z 97,A -100.0351,B 24.9374,C -1.8279,E1 24.9844,E2 185.3454} C_DIS
LIN {X -11.8678,Y -93.7104,Z 97,A -101.8557,B 24.9368,C -1.8366,E1 24.9794,E2 187.1466} C_DIS
LIN {X -14.7543,Y -93.2997,Z 97,A -103.8775,B 24.9373,C -1.8283,E1 24.9738,E2 189.1897} C_DIS
LIN {X -18.142,Y -92.7004,Z 97,A -105.8672,B 24.9371,C -1.8324,E1 24.9683,E2 191.1719} C_DIS
LIN {X -20.7449,Y -92.1539,Z 97,A -107.9846,B 24.9382,C -1.816,E1 24.9624,E2 193.3308} C_DIS
LIN {X -23.9068,Y -91.384,Z 97,A -109.5719,B 24.9372,C -1.8302,E1 24.9582,E2 194.8867} C_DIS
LIN {X -26.7175,Y -90.6014,Z 97,A -111.313,B 24.9371,C -1.8324,E1 24.9536,E2 196.6255} C_DIS
LIN {X -30.1277,Y -89.5251,Z 97,A -113.4384,B 24.9368,C -1.8355,E1 24.9479,E2 198.7472} C_DIS
LIN {X -33.4855,Y -88.324,Z 97,A -115.6283,B 24.9368,C -1.8366,E1 24.9422,E2 200.9392} C_DIS
LIN {X -36.8677,Y -86.9668,Z 97,A -117.8664,B 24.9367,C -1.8379,E1 24.9364,E2 203.1791} C_DIS
LIN {X -40.4049,Y -85.3825,Z 97,A -120.2829,B 24.9367,C -1.8383,E1 24.9303,E2 205.6005} C_DIS
LIN {X -42.786,Y -84.213,Z 97,A -122.3013,B 24.9374,C -1.8269,E1 24.9252,E2 207.6516} C_DIS
LIN {X -45.8233,Y -82.5997,Z 97,A -123.9075,B 24.9362,C -1.8455,E1 24.9213,E2 209.2182} C_DIS
LIN {X -48.8849,Y -80.8252,Z 97,A -126.0691,B 24.936,C -1.8481,E1 24.9161,E2 211.3801} C_DIS
LIN {X -51.9848,Y -78.8669,Z 97,A -128.2807,B 24.9357,C -1.8519,E1 24.9109,E2 213.5897} C_DIS
LIN {X -55.4773,Y -76.4516,Z 97,A -130.7999,B 24.9353,C -1.858,E1 24.9052,E2 216.103} C_DIS
LIN {X -58.2422,Y -74.3669,Z 97,A -132.988,B 24.9353,C -1.8589,E1 24.9003,E2 218.297} C_DIS
LIN {X -60.4249,Y -72.6034,Z 97,A -134.711,B 24.9351,C -1.8614,E1 24.8966,E2 220.0206} C_DIS
LIN {X -63.0827,Y -70.3065,Z 97,A -137.0812,B 24.9353,C -1.8578,E1 24.8916,E2 222.4086} C_DIS
LIN {X -66.2648,Y -67.3158,Z 97,A -139.4544,B 24.9343,C -1.8722,E1 24.8869,E2 224.7576} C_DIS
LIN {X -68.6237,Y -64.9098,Z 97,A -141.5266,B 24.934,C -1.8757,E1 24.8829,E2 226.8304} C_DIS
LIN {X -71.5884,Y -61.6258,Z 97,A -144.2916,B 24.9338,C -1.8791,E1 24.8777,E2 229.5995} C_DIS
LIN {X -73.8149,Y -58.9406,Z 97,A -146.437,B 24.9335,C -1.8831,E1 24.874,E2 231.7454} C_DIS
LIN {X -76.0866,Y -55.9758,Z 97,A -148.6532,B 24.933,C -1.8902,E1 24.8702,E2 233.9552} C_DIS
LIN {X -78.186,Y -53.0035,Z 97,A -150.8082,B 24.9325,C -1.8974,E1 24.8668,E2 236.1036} C_DIS
LIN {X -80.1785,Y -49.9383,Z 97,A -153.0032,B 24.932,C -1.9039,E1 24.8635,E2 238.2944} C_DIS
LIN {X -81.9295,Y -47.0103,Z 97,A -155.2348,B 24.932,C -1.9043,E1 24.8604,E2 240.5367} C_DIS
LIN {X -83.8964,Y -43.4054,Z 97,A -157.6335,B 24.9313,C -1.914,E1 24.8572,E2 242.925} C_DIS
LIN {X -85.3082,Y -40.5595,Z 97,A -159.7813,B 24.9314,C -1.9124,E1 24.8546,E2 245.0881} C_DIS
LIN {X -86.976,Y -36.8459,Z 97,A -162.0414,B 24.9305,C -1.926,E1 24.8521,E2 247.3282} C_DIS
LIN {X -88.0774,Y -34.1317,Z 97,A -163.9692,B 24.9305,C -1.9264,E1 24.8501,E2 249.2658} C_DIS
LIN {X -89.2583,Y -30.9114,Z 97,A -165.9126,B 24.9297,C -1.9369,E1 24.8483,E2 251.1953} C_DIS
LIN {X -90.4246,Y -27.3135,Z 97,A -168.357,B 24.9295,C -1.9391,E1 24.8462,E2 253.6485} C_DIS
LIN {X -91.3931,Y -23.8714,Z 97,A -170.4039,B 24.9287,C -1.9495,E1 24.8447,E2 255.6825} C_DIS
LIN {X -92.1454,Y -20.7816,Z 97,A -172.6186,B 24.929,C -1.9465,E1 24.8433,E2 257.9172} C_DIS
LIN {X -92.8477,Y -17.3767,Z 97,A -175.7256,B 24.9307,C -1.9226,E1 24.8417,E2 261.0998} C_DIS
LIN {X -93.7463,Y -11.5905,Z 97,A -178.4186,B 24.928,C -1.9599,E1 24.8407,E2 263.7198} C_DIS
LIN {X -94.2402,Y -6.4194,Z 97,A 178.6884,B 24.9266,C -1.9779,E1 24.8401,E2 266.5872} C_DIS
LIN {X -94.4359,Y -2.0961,Z 97,A 176.1161,B 24.9259,C -1.9879,E1 24.8398,E2 269.1511} C_DIS
LIN {X -94.4573,Y 0.5733,Z 97,A 173.6393,B 24.9275,C -1.9669,E1 24.8398,E2 271.6931} C_DIS
LIN {X -94.3249,Y 5.0256,Z 97,A 170.4985,B 24.9278,C -1.9623,E1 24.8404,E2 274.8636} C_DIS
LIN {X -93.8221,Y 10.9467,Z 97,A 168.3761,B 24.9236,C -2.0191,E1 24.8409,E2 276.8632} C_DIS
LIN {X -93.5415,Y 13.1314,Z 97,A 166.6453,B 24.9242,C -2.0112,E1 24.8416,E2 278.6233} C_DIS
LIN {X -92.9482,Y 16.8241,Z 97,A 164.5141,B 24.9233,C -2.0227,E1 24.8426,E2 280.7396} C_DIS
LIN {X -92.3192,Y 19.9901,Z 97,A 162.4986,B 24.9229,C -2.0271,E1 24.8437,E2 282.7564} C_DIS
LIN {X -91.5663,Y 23.1978,Z 97,A 160.4647,B 24.9225,C -2.0324,E1 24.8451,E2 284.7897} C_DIS
LIN {X -90.4391,Y 27.2647,Z 97,A 157.7867,B 24.9222,C -2.0368,E1 24.8471,E2 287.4727} C_DIS
LIN {X -89.3059,Y 30.7759,Z 97,A 155.1567,B 24.9226,C -2.0317,E1 24.8495,E2 290.13} C_DIS
LIN {X -88.1613,Y 33.9151,Z 97,A 153.5706,B 24.9211,C -2.0514,E1 24.851,E2 291.6778} C_DIS
LIN {X -87.024,Y 36.7319,Z 97,A 151.7055,B 24.9207,C -2.0564,E1 24.853,E2 293.5415} C_DIS
LIN {X -85.6659,Y 39.7967,Z 97,A 149.6967,B 24.9202,C -2.0633,E1 24.8553,E2 295.5449} C_DIS
LIN {X -84.1251,Y 42.9578,Z 97,A 147.286,B 24.9203,C -2.061,E1 24.8584,E2 297.974} C_DIS
LIN {X -82.0142,Y 46.863,Z 97,A 144.8218,B 24.9192,C -2.0759,E1 24.8617,E2 300.4156} C_DIS
LIN {X -79.4742,Y 51.0515,Z 97,A 141.8524,B 24.9185,C -2.0844,E1 24.866,E2 303.3799} C_DIS
LIN {X -77.4987,Y 54.0035,Z 97,A 139.7037,B 24.918,C -2.0905,E1 24.8694,E2 305.5246} C_DIS
LIN {X -75.6645,Y 56.5451,Z 97,A 137.895,B 24.9174,C -2.0985,E1 24.8724,E2 307.3229} C_DIS
LIN {X -71.8491,Y 61.3199,Z 97,A 134.1118,B 24.9168,C -2.1058,E1 24.879,E2 311.1063} C_DIS
LIN {X -69.7733,Y 63.6724,Z 97,A 132.1393,B 24.9166,C -2.1085,E1 24.8827,E2 313.0814} C_DIS
LIN {X -67.6327,Y 65.9433,Z 97,A 129.4584,B 24.9182,C -2.0884,E1 24.888,E2 315.8216} C_DIS
LIN {X -64.5673,Y 68.9458,Z 97,A 127.762,B 24.9155,C -2.123,E1 24.8913,E2 317.4426} C_DIS
LIN {X -62.3232,Y 70.9809,Z 97,A 125.7657,B 24.9155,C -2.1222,E1 24.8955,E2 319.4489} C_DIS
LIN {X -59.7168,Y 73.1875,Z 97,A 122.8779,B 24.9172,C -2.101,E1 24.9019,E2 322.398} C_DIS
LIN {X -56.1634,Y 75.9492,Z 97,A 120.9072,B 24.9149,C -2.1306,E1 24.9061,E2 324.3052} C_DIS
LIN {X -52.7045,Y 78.3884,Z 97,A 118.4299,B 24.9142,C -2.1386,E1 24.9118,E2 326.7719} C_DIS
LIN {X -50.2409,Y 79.9895,Z 97,A 116.5324,B 24.9142,C -2.1383,E1 24.9163,E2 328.6762} C_DIS
LIN {X -47.9407,Y 81.3887,Z 97,A 113.6469,B 24.9172,C -2.1014,E1 24.9235,E2 331.6581} C_DIS
LIN {X -42.471,Y 84.3739,Z 97,A 111.0335,B 24.9137,C -2.1448,E1 24.9297,E2 334.1755} C_DIS
LIN {X -40.229,Y 85.4646,Z 97,A 109.3851,B 24.9139,C -2.1427,E1 24.9339,E2 335.833} C_DIS
LIN {X -36.6671,Y 87.0513,Z 97,A 107.1818,B 24.9132,C -2.1514,E1 24.9395,E2 338.0208} C_DIS
LIN {X -33.5827,Y 88.2872,Z 97,A 105.1889,B 24.9129,C -2.1549,E1 24.9447,E2 340.0097} C_DIS
LIN {X -30.5097,Y 89.396,Z 97,A 102.7557,B 24.9139,C -2.1426,E1 24.9512,E2 342.4768} C_DIS
LIN {X -27.292,Y 90.4309,Z 97,A 100.9183,B 24.9132,C -2.1518,E1 24.956,E2 344.2954} C_DIS
LIN {X -23.3548,Y 91.5259,Z 97,A 98.6082,B 24.9125,C -2.1599,E1 24.9622,E2 346.5898} C_DIS
LIN {X -17.7242,Y 92.7808,Z 97,A 95.1357,B 24.9122,C -2.1638,E1 24.9717,E2 350.0573} C_DIS
LIN {X -14.3181,Y 93.3671,Z 97,A 93.052,B 24.912,C -2.1657,E1 24.9774,E2 352.1384} C_DIS
LIN {X -11.1609,Y 93.797,Z 97,A 91.1289,B 24.912,C -2.1671,E1 24.9827,E2 354.0593} C_DIS
LIN {X -7.426,Y 94.1662,Z 97,A 88.8074,B 24.912,C -2.1667,E1 24.9892,E2 356.383} C_DIS
LIN {X -4.0442,Y 94.3719,Z 97,A 86.7819,B 24.9118,C -2.1685,E1 24.9948,E2 358.4049} C_DIS
LIN {X -0.713,Y 94.4559,Z 97,A 84.8357,B 24.9116,C -2.1715,E1 25.0003,E2 360.3439} C_DIS
LIN {X 2.6307,Y 94.4223,Z 97,A 82.8099,B 24.9116,C -2.1719,E1 25.0059,E2 362.3686} C_DIS
LIN {X 5.9407,Y 94.2725,Z 97,A 80.7397,B 24.9116,C -2.1699,E1 25.0117,E2 364.4429} C_DIS
LIN {X 9.3831,Y 93.9924,Z 97,A 78.6117,B 24.9118,C -2.1685,E1 25.0176,E2 366.5728} C_DIS
LIN {X 12.8855,Y 93.5764,Z 97,A 76.5266,B 24.9117,C -2.1699,E1 25.0234,E2 368.6529} C_DIS
LIN {X 17.2109,Y 92.8787,Z 97,A 73.4537,B 24.9129,C -2.1547,E1 25.0319,E2 371.7585} C_DIS
LIN {X 21.8351,Y 91.9016,Z 97,A 70.9145,B 24.9121,C -2.1645,E1 25.0388,E2 374.271} C_DIS
LIN {X 25.6874,Y 90.8987,Z 97,A 68.5971,B 24.912,C -2.1664,E1 25.045,E2 376.5804} C_DIS
LIN {X 29.0807,Y 89.8706,Z 97,A 66.4477,B 24.9121,C -2.1648,E1 25.0507,E2 378.7297} C_DIS
LIN {X 32.473,Y 88.7014,Z 97,A 64.2702,B 24.9123,C -2.1628,E1 25.0565,E2 380.9075} C_DIS
LIN {X 35.3923,Y 87.5777,Z 97,A 62.2907,B 24.9127,C -2.158,E1 25.0616,E2 382.8938} C_DIS
LIN {X 38.9532,Y 86.0528,Z 97,A 60.2643,B 24.9119,C -2.1668,E1 25.0667,E2 384.8945} C_DIS
LIN {X 42.4983,Y 84.36,Z 97,A 57.4818,B 24.9133,C -2.1497,E1 25.0738,E2 387.7101} C_DIS
LIN {X 46.0405,Y 82.4784,Z 97,A 55.2541,B 24.913,C -2.1537,E1 25.0792,E2 389.9219} C_DIS
LIN {X 49.0649,Y 80.7158,Z 97,A 53.1351,B 24.9132,C -2.1508,E1 25.0843,E2 392.0414} C_DIS
LIN {X 52.3902,Y 78.5996,Z 97,A 50.6414,B 24.9138,C -2.1433,E1 25.0902,E2 394.5447} C_DIS
LIN {X 54.5755,Y 77.0976,Z 97,A 49.011,B 24.9141,C -2.1398,E1 25.0939,E2 396.1777} C_DIS
LIN {X 57.7054,Y 74.783,Z 97,A 46.7601,B 24.9141,C -2.1396,E1 25.0989,E2 398.4209} C_DIS
LIN {X 60.4219,Y 72.6059,Z 97,A 43.7278,B 24.9171,C -2.1026,E1 25.1056,E2 401.5291} C_DIS
LIN {X 64.2371,Y 69.2551,Z 97,A 41.5278,B 24.9151,C -2.128,E1 25.11,E2 403.6602} C_DIS
LIN {X 66.7442,Y 66.8422,Z 97,A 39.209,B 24.916,C -2.116,E1 25.1146,E2 405.9976} C_DIS
LIN {X 69.7361,Y 63.7128,Z 97,A 36.8779,B 24.9156,C -2.1209,E1 25.119,E2 408.3068} C_DIS
LIN {X 71.8404,Y 61.3301,Z 97,A 34.8418,B 24.9163,C -2.1126,E1 25.1228,E2 410.3535} C_DIS
LIN {X 74.244,Y 58.3977,Z 97,A 32.8413,B 24.9159,C -2.1181,E1 25.1263,E2 412.3316} C_DIS
LIN {X 75.8712,Y 56.2699,Z 97,A 30.973,B 24.9169,C -2.1051,E1 25.1294,E2 414.2216} C_DIS
LIN {X 77.6991,Y 53.7151,Z 97,A 29.1609,B 24.9169,C -2.1038,E1 25.1323,E2 416.028} C_DIS
LIN {X 79.3562,Y 51.2354,Z 97,A 27.3573,B 24.9173,C -2.0993,E1 25.1351,E2 417.8331} C_DIS
LIN {X 81.42,Y 47.8877,Z 97,A 24.6696,B 24.9187,C -2.0819,E1 25.139,E2 420.5483} C_DIS
LIN {X 83.6901,Y 43.7999,Z 97,A 22.1052,B 24.9185,C -2.0842,E1 25.1424,E2 423.0939} C_DIS
LIN {X 85.3717,Y 40.4273,Z 97,A 19.6625,B 24.9195,C -2.0719,E1 25.1454,E2 425.5523} C_DIS
LIN {X 87.1052,Y 36.5392,Z 97,A 17.326,B 24.9194,C -2.0737,E1 25.1479,E2 427.8719} C_DIS
LIN {X 88.2745,Y 33.6162,Z 97,A 15.7412,B 24.9188,C -2.0803,E1 25.1495,E2 429.4324} C_DIS
LIN {X 89.0676,Y 31.4549,Z 97,A 13.3982,B 24.9219,C -2.0409,E1 25.1518,E2 431.8553} C_DIS
LIN {X 90.3334,Y 27.6121,Z 97,A 11.5761,B 24.9207,C -2.057,E1 25.1533,E2 433.629} C_DIS
LIN {X 91.2555,Y 24.3909,Z 97,A 9.6318,B 24.9209,C -2.0541,E1 25.1547,E2 435.5689} C_DIS
LIN {X 92.3955,Y 19.6401,Z 97,A 6.6027,B 24.9218,C -2.0425,E1 25.1566,E2 438.6079} C_DIS
LIN {X 93.0656,Y 16.1717,Z 97,A 4.4459,B 24.9223,C -2.0353,E1 25.1577,E2 440.7691} C_DIS
LIN {X 93.6074,Y 12.6632,Z 97,A 2.383,B 24.9226,C -2.0319,E1 25.1585,E2 442.8279} C_DIS
LIN {X 94.0023,Y 9.2885,Z 97,A 0.3298,B 24.9231,C -2.0256,E1 25.1591,E2 444.8836} C_DIS
LIN {X 94.2764,Y 5.8832,Z 97,A -1.7179,B 24.9235,C -2.0199,E1 25.1596,E2 446.9326} C_DIS
LIN {X 94.4156,Y 2.8463,Z 97,A -3.5744,B 24.924,C -2.0136,E1 25.1597,E2 448.793} C_DIS
LIN {X 94.4573,Y -0.5661,Z 97,A -5.5883,B 24.9243,C -2.009,E1 25.1597,E2 450.8057} C_DIS
LIN {X 94.3666,Y -4.1673,Z 97,A -7.811,B 24.925,C -2.0006,E1 25.1596,E2 453.0351} C_DIS
LIN {X 94.1051,Y -8.1791,Z 97,A -10.2852,B 24.9256,C -1.9914,E1 25.159,E2 455.5164} C_DIS
LIN {X 93.731,Y -11.7087,Z 97,A -12.3243,B 24.9258,C -1.9887,E1 25.1584,E2 457.5496} C_DIS
LIN {X 93.2486,Y -15.0785,Z 97,A -14.2033,B 24.9258,C -1.9891,E1 25.1576,E2 459.4166} C_DIS
LIN {X 92.5531,Y -18.8772,Z 97,A -16.6832,B 24.9268,C -1.9764,E1 25.1563,E2 461.912} C_DIS
LIN {X 92.0014,Y -21.4049,Z 97,A -18.362,B 24.9274,C -1.9673,E1 25.1553,E2 463.6025} C_DIS
LIN {X 91.0541,Y -25.1365,Z 97,A -20.6426,B 24.9278,C -1.9619,E1 25.1536,E2 465.8827} C_DIS
LIN {X 90.0762,Y -28.4417,Z 97,A -22.7284,B 24.9283,C -1.9556,E1 25.1519,E2 467.9716} C_DIS
LIN {X 88.9575,Y -31.7688,Z 97,A -24.8287,B 24.9287,C -1.95,E1 25.15,E2 470.0732} C_DIS
LIN {X 87.7497,Y -34.9659,Z 97,A -26.6722,B 24.9285,C -1.9523,E1 25.1482,E2 471.901} C_DIS
LIN {X 86.7577,Y -37.359,Z 97,A -28.463,B 24.9295,C -1.9392,E1 25.1462,E2 473.7129} C_DIS
LIN {X 85.7519,Y -39.6119,Z 97,A -30.3882,B 24.931,C -1.9187,E1 25.1439,E2 475.6762} C_DIS
LIN {X 84.2413,Y -42.7306,Z 97,A -31.9628,B 24.93,C -1.9322,E1 25.142,E2 477.2105} C_DIS
LIN {X 82.9565,Y -45.1737,Z 97,A -33.848,B 24.9309,C -1.9193,E1 25.1395,E2 479.1161} C_DIS
LIN {X 80.8641,Y -48.8209,Z 97,A -36.1038,B 24.9307,C -1.923,E1 25.1363,E2 481.3516} C_DIS
LIN {X 79.2003,Y -51.4783,Z 97,A -37.9164,B 24.9308,C -1.921,E1 25.1336,E2 483.16} C_DIS
LIN {X 77.9437,Y -53.3613,Z 97,A -39.8508,B 24.9326,C -1.8962,E1 25.1305,E2 485.1433} C_DIS
LIN {X 75.0906,Y -57.3063,Z 97,A -42.4141,B 24.9321,C -1.9027,E1 25.1262,E2 487.6791} C_DIS
LIN {X 73.3345,Y -59.5355,Z 97,A -44.4431,B 24.9333,C -1.8867,E1 25.1226,E2 489.7364} C_DIS
LIN {X 68.161,Y -65.3952,Z 97,A -48.7826,B 24.9331,C -1.8896,E1 25.1146,E2 494.0497} C_DIS
LIN {X 66.3374,Y -67.2441,Z 97,A -50.9249,B 24.9348,C -1.8648,E1 25.1102,E2 496.2415} C_DIS
LIN {X 63.642,Y -69.8012,Z 97,A -52.8504,B 24.9343,C -1.8716,E1 25.1063,E2 498.1433} C_DIS
LIN {X 60.4004,Y -72.6237,Z 97,A -55.1637,B 24.934,C -1.8765,E1 25.1014,E2 500.4358} C_DIS
LIN {X 57.7945,Y -74.7144,Z 97,A -57.0724,B 24.934,C -1.8765,E1 25.0972,E2 502.3375} C_DIS
LIN {X 54.8822,Y -76.8788,Z 97,A -59.3732,B 24.9346,C -1.8682,E1 25.092,E2 504.6498} C_DIS
LIN {X 52.1241,Y -78.7751,Z 97,A -61.4269,B 24.9349,C -1.8633,E1 25.0873,E2 506.7081} C_DIS
LIN {X 48.8024,Y -80.8754,Z 97,A -64.4569,B 24.9369,C -1.8354,E1 25.0799,E2 509.7946} C_DIS
LIN {X 45.3168,Y -82.8789,Z 97,A -66.2097,B 24.9354,C -1.8559,E1 25.0758,E2 511.4938} C_DIS
LIN {X 40.8548,Y -85.1663,Z 97,A -69.1941,B 24.9356,C -1.8529,E1 25.0683,E2 514.4771} C_DIS
LIN {X 38.395,Y -86.3043,Z 97,A -70.7614,B 24.9356,C -1.8532,E1 25.0644,E2 516.0399} C_DIS
LIN {X 34.9536,Y -87.7545,Z 97,A -73.1666,B 24.9362,C -1.8448,E1 25.0581,E2 518.4593} C_DIS
LIN {X 31.9474,Y -88.8931,Z 97,A -75.1314,B 24.9364,C -1.8417,E1 25.053,E2 520.4273} C_DIS
LIN {X 28.7562,Y -89.9756,Z 97,A -77.1494,B 24.9365,C -1.8402,E1 25.0476,E2 522.4451} C_DIS
LIN {X 25.5617,Y -90.9343,Z 97,A -79.2401,B 24.9368,C -1.8355,E1 25.042,E2 524.5434} C_DIS
LIN {X 20.6166,Y -92.1825,Z 97,A -82.304,B 24.937,C -1.8335,E1 25.0337,E2 527.6075} C_DIS
LIN {X 17.2652,Y -92.8689,Z 97,A -84.4265,B 24.9372,C -1.8301,E1 25.0278,E2 529.7356} C_DIS
LIN {X 13.4542,Y -93.4956,Z 97,A -86.6988,B 24.9372,C -1.8309,E1 25.0216,E2 532.0039} C_DIS
LIN {X 10.0916,Y -93.9183,Z 97,A -88.4194,B 24.9364,C -1.8415,E1 25.0169,E2 533.6981} C_DIS
LIN {X 7.5096,Y -94.1595,Z 97,A -90.2659,B 24.9372,C -1.831,E1 25.0117,E2 535.5683} C_DIS
LIN {X 3.9371,Y -94.3765,Z 97,A -92.4767,B 24.9373,C -1.8288,E1 25.0055,E2 537.7837} C_DIS
LIN {X 0.6825,Y -94.4556,Z 97,A -94.406,B 24.9373,C -1.8298,E1 25.0001,E2 539.7102} C_DIS
Enddeposition()
LIN {X 0.6825,Y -94.4556,Z 97,A -94.406,B 24.9373,C -1.8298,E1 25.0001,E2 539.7102} C_DIS
Startdeposition()
$VEL.CP = VEL_PRINT
LIN {X 1.7535,Y -93.5376,Z 97,A -92.9091,B 24.9341,C -1.8751,E1 25.0046,E2 538.106} C_DIS
LIN {X 5.1871,Y -93.4101,Z 97,A -90.8051,B 24.9341,C -1.8759,E1 25.0105,E2 536.0008} C_DIS
LIN {X 8.5483,Y -93.1627,Z 97,A -88.7267,B 24.9339,C -1.8774,E1 25.0163,E2 533.9199} C_DIS
LIN {X 11.9879,Y -92.7828,Z 97,A -86.6073,B 24.9339,C -1.8787,E1 25.0221,E2 531.799} C_DIS
LIN {X 15.4528,Y -92.269,Z 97,A -84.485,B 24.9338,C -1.8795,E1 25.028,E2 529.677} C_DIS
LIN {X 18.832,Y -91.639,Z 97,A -82.3799,B 24.9337,C -1.8812,E1 25.0338,E2 527.5702} C_DIS
LIN {X 22.2287,Y -90.8749,Z 97,A -80.2546,B 24.9335,C -1.883,E1 25.0395,E2 525.4437} C_DIS
LIN {X 25.547,Y -89.9984,Z 97,A -78.1595,B 24.9334,C -1.885,E1 25.0452,E2 523.3472} C_DIS
LIN {X 28.8323,Y -89.0003,Z 97,A -76.0624,B 24.9332,C -1.8873,E1 25.0508,E2 521.2486} C_DIS
LIN {X 32.0788,Y -87.8823,Z 97,A -73.9634,B 24.933,C -1.8899,E1 25.0563,E2 519.1477} C_DIS
LIN {X 35.2211,Y -86.6709,Z 97,A -71.8846,B 24.9328,C -1.8933,E1 25.0617,E2 517.0654} C_DIS
LIN {X 38.4068,Y -85.307,Z 97,A -69.7725,B 24.9326,C -1.8962,E1 25.0671,E2 514.9517} C_DIS
LIN {X 41.598,Y -83.7972,Z 97,A -67.6407,B 24.9324,C -1.8985,E1 25.0725,E2 512.82} C_DIS
LIN {X 44.5726,Y -82.2535,Z 97,A -65.5735,B 24.9321,C -1.9026,E1 25.0776,E2 510.749} C_DIS
LIN {X 47.5993,Y -80.5399,Z 97,A -63.4599,B 24.9319,C -1.9058,E1 25.0827,E2 508.6341} C_DIS
LIN {X 50.5039,Y -78.751,Z 97,A -61.37,B 24.9316,C -1.9098,E1 25.0877,E2 506.5414} C_DIS
LIN {X 53.3601,Y -76.8444,Z 97,A -59.2741,B 24.9313,C -1.9138,E1 25.0925,E2 504.4433} C_DIS
LIN {X 56.2251,Y -74.7736,Z 97,A -57.1437,B 24.9311,C -1.917,E1 25.0973,E2 502.3129} C_DIS
LIN {X 58.9006,Y -72.6848,Z 97,A -55.0626,B 24.9308,C -1.9216,E1 25.1019,E2 500.2286} C_DIS
LIN {X 61.5236,Y -70.4784,Z 97,A -52.9715,B 24.9305,C -1.9261,E1 25.1063,E2 498.1351} C_DIS
LIN {X 64.0597,Y -68.1815,Z 97,A -50.87,B 24.9301,C -1.9312,E1 25.1106,E2 496.03} C_DIS
LIN {X 66.5546,Y -65.7484,Z 97,A -48.7665,B 24.9298,C -1.9352,E1 25.1148,E2 493.9259} C_DIS
LIN {X 68.9134,Y -63.2716,Z 97,A -46.6797,B 24.9294,C -1.9402,E1 25.1188,E2 491.8365} C_DIS
LIN {X 71.1733,Y -60.7184,Z 97,A -44.581,B 24.929,C -1.9459,E1 25.1226,E2 489.7337} C_DIS
LIN {X 73.3986,Y -58.0087,Z 97,A -42.4713,B 24.9287,C -1.9502,E1 25.1263,E2 487.6237} C_DIS
LIN {X 75.4545,Y -55.3081,Z 97,A -40.3914,B 24.9283,C -1.9559,E1 25.1298,E2 485.5403} C_DIS
LIN {X 77.446,Y -52.4832,Z 97,A -38.2851,B 24.9279,C -1.9614,E1 25.1332,E2 483.4314} C_DIS
LIN {X 79.3285,Y -49.5918,Z 97,A -36.1901,B 24.9275,C -1.9667,E1 25.1363,E2 481.3344} C_DIS
LIN {X 81.128,Y -46.5899,Z 97,A -34.0735,B 24.9271,C -1.9718,E1 25.1393,E2 479.2165} C_DIS
LIN {X 82.7895,Y -43.569,Z 97,A -31.9819,B 24.9267,C -1.9773,E1 25.1421,E2 477.1231} C_DIS
LIN {X 84.2988,Y -40.5719,Z 97,A -29.9155,B 24.9262,C -1.9838,E1 25.1446,E2 475.0523} C_DIS
LIN {X 85.748,Y -37.4117,Z 97,A -27.7961,B 24.9258,C -1.9899,E1 25.1471,E2 472.9301} C_DIS
LIN {X 87.0939,Y -34.1616,Z 97,A -25.6837,B 24.9254,C -1.9949,E1 25.1493,E2 470.8175} C_DIS
LIN {X 88.2891,Y -30.9418,Z 97,A -23.5959,B 24.9249,C -2.0008,E1 25.1513,E2 468.7274} C_DIS
LIN {X 89.3462,Y -27.7419,Z 97,A -21.5242,B 24.9244,C -2.0076,E1 25.153,E2 466.6515} C_DIS
LIN {X 90.3211,Y -24.3813,Z 97,A -19.4143,B 24.924,C -2.0131,E1 25.1546,E2 464.5408} C_DIS
LIN {X 91.1402,Y -21.1147,Z 97,A -17.3534,B 24.9235,C -2.0196,E1 25.156,E2 462.4765} C_DIS
LIN {X 91.8308,Y -17.8746,Z 97,A -15.276,B 24.9229,C -2.0279,E1 25.1571,E2 460.3915} C_DIS
LIN {X 92.5435,Y -13.7254,Z 97,A -12.6681,B 24.9222,C -2.0373,E1 25.1583,E2 457.7769} C_DIS
LIN {X 92.9855,Y -10.3138,Z 97,A -10.576,B 24.9217,C -2.0435,E1 25.159,E2 455.6824} C_DIS
LIN {X 93.303,Y -6.8722,Z 97,A -8.4919,B 24.9213,C -2.0491,E1 25.1595,E2 453.5975} C_DIS
LIN {X 93.4917,Y -3.4595,Z 97,A -6.4098,B 24.9208,C -2.0554,E1 25.1597,E2 451.5129} C_DIS
LIN {X 93.5555,Y -0.1708,Z 97,A -4.5738,B 24.9208,C -2.0551,E1 25.1597,E2 449.6885} C_DIS
LIN {X 93.511,Y 2.8388,Z 97,A -2.665,B 24.9201,C -2.0635,E1 25.1597,E2 447.7712} C_DIS
LIN {X 93.3429,Y 6.2815,Z 97,A -0.5729,B 24.9197,C -2.0696,E1 25.1593,E2 445.6773} C_DIS
LIN {X 93.0423,Y 9.7717,Z 97,A 1.5383,B 24.9193,C -2.0751,E1 25.1588,E2 443.5656} C_DIS
LIN {X 92.6227,Y 13.1678,Z 97,A 3.6303,B 24.9187,C -2.0816,E1 25.158,E2 441.4706} C_DIS
LIN {X 92.0705,Y 16.5948,Z 97,A 5.7305,B 24.9183,C -2.0873,E1 25.157,E2 439.3693} C_DIS
LIN {X 91.4121,Y 19.9047,Z 97,A 7.8141,B 24.9177,C -2.0943,E1 25.1558,E2 437.2812} C_DIS
LIN {X 90.5991,Y 23.3273,Z 97,A 9.9216,B 24.9174,C -2.0991,E1 25.1544,E2 435.1745} C_DIS
LIN {X 89.7036,Y 26.5636,Z 97,A 11.9887,B 24.9168,C -2.1058,E1 25.1528,E2 433.1036} C_DIS
LIN {X 88.6524,Y 29.8849,Z 97,A 14.0921,B 24.9164,C -2.111,E1 25.151,E2 430.9997} C_DIS
LIN {X 87.5009,Y 33.1051,Z 97,A 16.1875,B 24.9159,C -2.1172,E1 25.149,E2 428.9013} C_DIS
LIN {X 86.2013,Y 36.3551,Z 97,A 18.2983,B 24.9155,C -2.1222,E1 25.1468,E2 426.7904} C_DIS
LIN {X 84.8361,Y 39.4359,Z 97,A 20.3762,B 24.915,C -2.1286,E1 25.1444,E2 424.7087} C_DIS
LIN {X 83.32,Y 42.5456,Z 97,A 22.4765,B 24.9146,C -2.1338,E1 25.1417,E2 422.6073} C_DIS
LIN {X 81.7381,Y 45.5111,Z 97,A 24.5518,B 24.9141,C -2.14,E1 25.139,E2 420.5282} C_DIS
LIN {X 79.9645,Y 48.5596,Z 97,A 26.6693,B 24.9138,C -2.1442,E1 25.1359,E2 418.4118} C_DIS
LIN {X 78.0926,Y 51.5161,Z 97,A 28.7827,B 24.9134,C -2.1486,E1 25.1327,E2 416.2985} C_DIS
LIN {X 76.1757,Y 54.3105,Z 97,A 30.8651,B 24.913,C -2.1541,E1 25.1294,E2 414.2133} C_DIS
LIN {X 74.1022,Y 57.1072,Z 97,A 32.9736,B 24.9126,C -2.1584,E1 25.1259,E2 412.1046} C_DIS
LIN {X 71.9596,Y 59.7844,Z 97,A 35.0681,B 24.9122,C -2.1632,E1 25.1222,E2 410.0086} C_DIS
LIN {X 69.705,Y 62.3985,Z 97,A 37.1688,B 24.9119,C -2.1675,E1 25.1183,E2 407.9071} C_DIS
LIN {X 67.3644,Y 64.9184,Z 97,A 39.2697,B 24.9115,C -2.1719,E1 25.1143,E2 405.8048} C_DIS
LIN {X 64.9275,Y 67.3556,Z 97,A 41.3654,B 24.9112,C -2.1758,E1 25.1101,E2 403.7088} C_DIS
LIN {X 62.4191,Y 69.6866,Z 97,A 43.4554,B 24.9109,C -2.1798,E1 25.1058,E2 401.6178} C_DIS
LIN {X 59.8329,Y 71.9193,Z 97,A 45.554,B 24.9105,C -2.1841,E1 25.1013,E2 399.5173} C_DIS
LIN {X 57.102,Y 74.1061,Z 97,A 47.6705,B 24.9103,C -2.187,E1 25.0967,E2 397.4017} C_DIS
LIN {X 54.3237,Y 76.1662,Z 97,A 49.7768,B 24.91,C -2.1903,E1 25.0919,E2 395.2951} C_DIS
LIN {X 51.5287,Y 78.0843,Z 97,A 51.8677,B 24.9097,C -2.1942,E1 25.0871,E2 393.2021} C_DIS
LIN {X 48.5561,Y 79.9666,Z 97,A 53.9876,B 24.9095,C -2.1962,E1 25.082,E2 391.084} C_DIS
LIN {X 45.588,Y 81.6951,Z 97,A 56.0863,B 24.9093,C -2.199,E1 25.0769,E2 388.985} C_DIS
LIN {X 42.5474,Y 83.3192,Z 97,A 58.1852,B 24.9091,C -2.2014,E1 25.0718,E2 386.8865} C_DIS
LIN {X 39.5641,Y 84.7765,Z 97,A 60.1553,B 24.9091,C -2.2016,E1 25.0668,E2 384.921} C_DIS
LIN {X 36.8656,Y 85.9861,Z 97,A 62.1546,B 24.9084,C -2.2102,E1 25.0617,E2 382.9061} C_DIS
LIN {X 33.6672,Y 87.288,Z 97,A 64.2446,B 24.9083,C -2.2114,E1 25.0562,E2 380.8178} C_DIS
LIN {X 30.5216,Y 88.4365,Z 97,A 66.2985,B 24.9081,C -2.2134,E1 25.0508,E2 378.7635} C_DIS
LIN {X 27.1711,Y 89.5232,Z 97,A 68.4429,B 24.9081,C -2.2146,E1 25.0451,E2 376.6202} C_DIS
LIN {X 23.8389,Y 90.4676,Z 97,A 70.5618,B 24.9079,C -2.2159,E1 25.0394,E2 374.5016} C_DIS
LIN {X 20.5106,Y 91.2797,Z 97,A 72.6557,B 24.9079,C -2.2169,E1 25.0337,E2 372.4082} C_DIS
LIN {X 17.1572,Y 91.9689,Z 97,A 74.7961,B 24.9076,C -2.2193,E1 25.0278,E2 370.2647} C_DIS
LIN {X 13.7333,Y 92.5423,Z 97,A 76.6685,B 24.9083,C -2.2111,E1 25.0227,E2 368.4133} C_DIS
LIN {X 9.7697,Y 93.0425,Z 97,A 79.2361,B 24.9079,C -2.2158,E1 25.0156,E2 365.8366} C_DIS
LIN {X 6.2788,Y 93.3431,Z 97,A 81.362,B 24.9079,C -2.2152,E1 25.0097,E2 363.7132} C_DIS
LIN {X 2.8447,Y 93.5108,Z 97,A 83.469,B 24.9079,C -2.2152,E1 25.0038,E2 361.607} C_DIS
LIN {X -0.5425,Y 93.5525,Z 97,A 85.5655,B 24.9079,C -2.2155,E1 24.9979,E2 359.5098} C_DIS
LIN {X -3.9848,Y 93.4691,Z 97,A 87.6708,B 24.9079,C -2.2147,E1 24.9921,E2 357.406} C_DIS
LIN {X -7.4806,Y 93.2545,Z 97,A 89.8018,B 24.9081,C -2.2133,E1 24.9861,E2 355.2774} C_DIS
LIN {X -10.8366,Y 92.9243,Z 97,A 91.8917,B 24.9081,C -2.2131,E1 24.9803,E2 353.1869} C_DIS
LIN {X -14.2618,Y 92.4606,Z 97,A 94.009,B 24.9082,C -2.2117,E1 24.9745,E2 351.0711} C_DIS
LIN {X -17.6495,Y 91.8741,Z 97,A 96.1327,B 24.9083,C -2.2107,E1 24.9686,E2 348.9476} C_DIS
LIN {X -21.0999,Y 91.1436,Z 97,A 98.2588,B 24.9086,C -2.2077,E1 24.9629,E2 346.8261} C_DIS
LIN {X -24.3532,Y 90.3287,Z 97,A 100.3423,B 24.9086,C -2.2066,E1 24.9572,E2 344.7421} C_DIS
LIN {X -27.6941,Y 89.361,Z 97,A 102.4621,B 24.9089,C -2.2039,E1 24.9516,E2 342.6251} C_DIS
LIN {X -30.8574,Y 88.3187,Z 97,A 104.4509,B 24.9092,C -2.1997,E1 24.9463,E2 340.6424} C_DIS
LIN {X -33.6658,Y 87.2886,Z 97,A 106.4476,B 24.909,C -2.2027,E1 24.9411,E2 338.6345} C_DIS
LIN {X -36.8493,Y 85.9931,Z 97,A 108.5578,B 24.9092,C -2.1999,E1 24.9356,E2 336.5262} C_DIS
LIN {X -40.0035,Y 84.5719,Z 97,A 110.6995,B 24.9094,C -2.1974,E1 24.9302,E2 334.3851} C_DIS
LIN {X -43.0646,Y 83.0548,Z 97,A 112.7777,B 24.9097,C -2.1935,E1 24.9251,E2 332.3105} C_DIS
LIN {X -46.062,Y 81.4305,Z 97,A 114.8808,B 24.91,C -2.1904,E1 24.9199,E2 330.2087} C_DIS
LIN {X -49.0687,Y 79.6551,Z 97,A 117.031,B 24.9103,C -2.1869,E1 24.9148,E2 328.0603} C_DIS
LIN {X -51.9746,Y 77.7903,Z 97,A 119.1573,B 24.9106,C -2.1832,E1 24.9098,E2 325.9358} C_DIS
LIN {X -54.8037,Y 75.8237,Z 97,A 121.2862,B 24.9109,C -2.1796,E1 24.905,E2 323.8083} C_DIS
LIN {X -57.5344,Y 73.7729,Z 97,A 123.3746,B 24.9113,C -2.175,E1 24.9004,E2 321.723} C_DIS
LIN {X -60.2317,Y 71.5879,Z 97,A 125.5182,B 24.9116,C -2.1709,E1 24.8958,E2 319.5811} C_DIS
LIN {X -62.6192,Y 69.5074,Z 97,A 127.3997,B 24.9121,C -2.1647,E1 24.8919,E2 317.7069} C_DIS
LIN {X -65.0276,Y 67.2591,Z 97,A 129.3476,B 24.9127,C -2.1577,E1 24.8879,E2 315.7676} C_DIS
LIN {X -67.3585,Y 64.9245,Z 97,A 131.419,B 24.9129,C -2.1544,E1 24.8839,E2 313.6952} C_DIS
LIN {X -69.6977,Y 62.4066,Z 97,A 133.4927,B 24.9134,C -2.1482,E1 24.88,E2 311.6272} C_DIS
LIN {X -71.7364,Y 60.053,Z 97,A 135.5154,B 24.9135,C -2.1469,E1 24.8763,E2 309.5983} C_DIS
LIN {X -73.8356,Y 57.4531,Z 97,A 137.5545,B 24.914,C -2.1413,E1 24.8728,E2 307.5631} C_DIS
LIN {X -75.8193,Y 54.8098,Z 97,A 139.6675,B 24.9142,C -2.1386,E1 24.8693,E2 305.4463} C_DIS
LIN {X -77.7866,Y 51.98,Z 97,A 141.7864,B 24.9147,C -2.133,E1 24.866,E2 303.3301} C_DIS
LIN {X -79.6163,Y 49.1312,Z 97,A 143.8623,B 24.9151,C -2.1272,E1 24.8629,E2 301.2575} C_DIS
LIN {X -81.4047,Y 46.1081,Z 97,A 146.0455,B 24.9155,C -2.1221,E1 24.8598,E2 299.0753} C_DIS
LIN {X -83.0537,Y 43.0668,Z 97,A 148.1512,B 24.9161,C -2.1154,E1 24.8571,E2 296.9742} C_DIS
LIN {X -84.5764,Y 39.9938,Z 97,A 150.2847,B 24.9165,C -2.1102,E1 24.8545,E2 294.8416} C_DIS
LIN {X -85.9858,Y 36.8662,Z 97,A 152.3999,B 24.917,C -2.1043,E1 24.8521,E2 292.7288} C_DIS
LIN {X -87.2792,Y 33.6898,Z 97,A 154.4945,B 24.9175,C -2.0977,E1 24.85,E2 290.6382} C_DIS
LIN {X -88.4542,Y 30.4712,Z 97,A 156.6164,B 24.9179,C -2.092,E1 24.848,E2 288.518} C_DIS
LIN {X -89.5262,Y 27.1615,Z 97,A 158.7637,B 24.9184,C -2.0858,E1 24.8462,E2 286.373} C_DIS
LIN {X -90.4687,Y 23.8346,Z 97,A 160.8886,B 24.9189,C -2.0794,E1 24.8447,E2 284.2511} C_DIS
LIN {X -91.2823,Y 20.4993,Z 97,A 163.0076,B 24.9194,C -2.0732,E1 24.8433,E2 282.1344} C_DIS
LIN {X -91.9729,Y 17.1365,Z 97,A 165.1225,B 24.9199,C -2.0669,E1 24.8422,E2 280.0222} C_DIS
LIN {X -92.5394,Y 13.752,Z 97,A 167.2532,B 24.9203,C -2.0611,E1 24.8413,E2 277.8926} C_DIS
LIN {X -92.9836,Y 10.3307,Z 97,A 169.374,B 24.9208,C -2.0545,E1 24.8406,E2 275.7748} C_DIS
LIN {X -93.294,Y 6.9868,Z 97,A 171.4528,B 24.9213,C -2.0486,E1 24.8401,E2 273.6976} C_DIS
LIN {X -93.4913,Y 3.4702,Z 97,A 173.6242,B 24.9218,C -2.0421,E1 24.8398,E2 271.5286} C_DIS
LIN {X -93.5565,Y -0.0091,Z 97,A 175.7961,B 24.9222,C -2.0365,E1 24.8398,E2 269.357} C_DIS
LIN {X -93.493,Y -3.4229,Z 97,A 177.8755,B 24.9228,C -2.0295,E1 24.84,E2 267.2818} C_DIS
LIN {X -93.3063,Y -6.8232,Z 97,A 179.946,B 24.9233,C -2.0224,E1 24.8403,E2 265.2158} C_DIS
LIN {X -92.991,Y -10.2621,Z 97,A -177.9002,B 24.9237,C -2.0169,E1 24.8409,E2 263.0623} C_DIS
LIN {X -92.5468,Y -13.7021,Z 97,A -175.7573,B 24.9242,C -2.0108,E1 24.8418,E2 260.9212} C_DIS
LIN {X -91.975,Y -17.1254,Z 97,A -173.6085,B 24.9246,C -2.0049,E1 24.8428,E2 258.7737} C_DIS
LIN {X -91.2812,Y -20.5042,Z 97,A -171.4818,B 24.9251,C -1.9988,E1 24.8441,E2 256.649} C_DIS
LIN {X -90.4668,Y -23.8419,Z 97,A -169.3625,B 24.9255,C -1.9928,E1 24.8455,E2 254.5316} C_DIS
LIN {X -89.5304,Y -27.1474,Z 97,A -167.246,B 24.926,C -1.9869,E1 24.8472,E2 252.4171} C_DIS
LIN {X -88.4664,Y -30.4367,Z 97,A -165.1129,B 24.9264,C -1.9811,E1 24.8491,E2 250.2856} C_DIS
LIN {X -87.2882,Y -33.6669,Z 97,A -163.0102,B 24.9269,C -1.9748,E1 24.8512,E2 248.1861} C_DIS
LIN {X -85.9985,Y -36.8363,Z 97,A -160.8972,B 24.9273,C -1.9693,E1 24.8535,E2 246.0743} C_DIS
LIN {X -84.5692,Y -40.009,Z 97,A -158.7425,B 24.9277,C -1.9641,E1 24.856,E2 243.9205} C_DIS
LIN {X -83.046,Y -43.0818,Z 97,A -156.645,B 24.9281,C -1.9582,E1 24.8586,E2 241.8257} C_DIS
LIN {X -81.4013,Y -46.1141,Z 97,A -154.5012,B 24.9285,C -1.9535,E1 24.8615,E2 239.6819} C_DIS
LIN {X -79.6521,Y -49.0737,Z 97,A -152.4009,B 24.9289,C -1.9478,E1 24.8646,E2 237.5844} C_DIS
LIN {X -77.9587,Y -51.7192,Z 97,A -150.7373,B 24.9298,C -1.9346,E1 24.8671,E2 235.944} C_DIS
LIN {X -76.4858,Y -53.8758,Z 97,A -148.842,B 24.9294,C -1.94,E1 24.8701,E2 234.0264} C_DIS
LIN {X -74.4568,Y -56.6469,Z 97,A -146.7343,B 24.9298,C -1.935,E1 24.8737,E2 231.9204} C_DIS
LIN {X -72.3196,Y -59.3512,Z 97,A -144.6115,B 24.9301,C -1.9304,E1 24.8774,E2 229.7987} C_DIS
LIN {X -70.0774,Y -61.9825,Z 97,A -142.4872,B 24.9305,C -1.9258,E1 24.8813,E2 227.6758} C_DIS
LIN {X -67.7568,Y -64.5112,Z 97,A -140.3721,B 24.9308,C -1.9216,E1 24.8853,E2 225.5614} C_DIS
LIN {X -65.3449,Y -66.9531,Z 97,A -138.2618,B 24.9311,C -1.9175,E1 24.8895,E2 223.4521} C_DIS
LIN {X -62.8459,Y -69.304,Z 97,A -136.1473,B 24.9313,C -1.9137,E1 24.8938,E2 221.338} C_DIS
LIN {X -60.2371,Y -71.5833,Z 97,A -134.0173,B 24.9316,C -1.9099,E1 24.8984,E2 219.2087} C_DIS
LIN {X -57.5633,Y -73.7506,Z 97,A -131.9123,B 24.9319,C -1.906,E1 24.903,E2 217.1053} C_DIS
LIN {X -54.8063,Y -75.8218,Z 97,A -129.7705,B 24.9321,C -1.9033,E1 24.9078,E2 214.9622} C_DIS
LIN {X -51.9714,Y -77.7924,Z 97,A -127.6534,B 24.9323,C -1.9,E1 24.9127,E2 212.846} C_DIS
LIN {X -49.0797,Y -79.6484,Z 97,A -125.5574,B 24.9326,C -1.8965,E1 24.9176,E2 210.7516} C_DIS
LIN {X -46.1218,Y -81.3969,Z 97,A -123.4305,B 24.9327,C -1.8943,E1 24.9228,E2 208.6236} C_DIS
LIN {X -43.1128,Y -83.0298,Z 97,A -121.3417,B 24.9329,C -1.8913,E1 24.9279,E2 206.5361} C_DIS
LIN {X -40.0055,Y -84.5709,Z 97,A -119.1937,B 24.9331,C -1.8896,E1 24.9333,E2 204.3867} C_DIS
LIN {X -36.8564,Y -85.99,Z 97,A -117.0774,B 24.9332,C -1.8873,E1 24.9387,E2 202.2708} C_DIS
LIN {X -33.674,Y -87.2854,Z 97,A -114.9851,B 24.9334,C -1.8849,E1 24.9442,E2 200.1797} C_DIS
LIN {X -30.4463,Y -88.463,Z 97,A -112.8787,B 24.9335,C -1.8832,E1 24.9497,E2 198.0732} C_DIS
LIN {X -27.1787,Y -89.5208,Z 97,A -110.7671,B 24.9336,C -1.8819,E1 24.9553,E2 195.9609} C_DIS
LIN {X -23.8558,Y -90.4631,Z 97,A -108.6551,B 24.9337,C -1.8805,E1 24.961,E2 193.8491} C_DIS
LIN {X -20.5318,Y -91.2748,Z 97,A -106.55,B 24.9337,C -1.8797,E1 24.9668,E2 191.743} C_DIS
LIN {X -17.1296,Y -91.9742,Z 97,A -104.4249,B 24.9338,C -1.8788,E1 24.9726,E2 189.6177} C_DIS
LIN {X -13.7373,Y -92.5417,Z 97,A -102.2972,B 24.9338,C -1.879,E1 24.9785,E2 187.4877} C_DIS
LIN {X -10.3122,Y -92.9857,Z 97,A -100.1834,B 24.9338,C -1.8786,E1 24.9843,E2 185.3734} C_DIS
LIN {X -6.8885,Y -93.3018,Z 97,A -98.095,B 24.9338,C -1.878,E1 24.9901,E2 183.2856} C_DIS
LIN {X -3.446,Y -93.4923,Z 97,A -95.9798,B 24.9338,C -1.8783,E1 24.996,E2 181.1692} C_DIS
LIN {X 0.003,Y -93.5558,Z 97,A -93.8553,B 24.9338,C -1.8791,E1 25.002,E2 179.0426} C_DIS
LIN {X 0.003,Y -93.5558,Z 97,A -93.8553,B 24.9338,C -1.8791,E1 25.002,E2 179.0426} C_DIS
Enddeposition()
LIN {X 0.6951,Y -100.835,Z 98,A -93.7868,B 24.9428,C -1.7477,E1 25.0013,E2 179.2857} C_DIS
Startdeposition()
$VEL.CP = VEL_PRINT
LIN {X 3.7116,Y -100.771,Z 98,A -91.695,B 24.9418,C -1.7626,E1 25.0072,E2 177.1591} C_DIS
LIN {X 6.2151,Y -100.6474,Z 98,A -90.3051,B 24.9418,C -1.7619,E1 25.0111,E2 175.7714} C_DIS
LIN {X 8.6517,Y -100.4675,Z 98,A -88.9017,B 24.9418,C -1.7631,E1 25.015,E2 174.3658} C_DIS
LIN {X 11.63,Y -100.1645,Z 98,A -87.287,B 24.9418,C -1.7608,E1 25.0195,E2 172.7576} C_DIS
LIN {X 14.7962,Y -99.7479,Z 98,A -85.3746,B 24.9416,C -1.7658,E1 25.0248,E2 170.8352} C_DIS
LIN {X 17.2708,Y -99.3491,Z 98,A -83.9854,B 24.9416,C -1.7655,E1 25.0286,E2 169.448} C_DIS
LIN {X 19.7037,Y -98.8953,Z 98,A -82.565,B 24.9415,C -1.7672,E1 25.0325,E2 168.0252} C_DIS
LIN {X 22.1248,Y -98.382,Z 98,A -81.1619,B 24.9414,C -1.7684,E1 25.0364,E2 166.6212} C_DIS
LIN {X 24.8566,Y -97.7261,Z 98,A -79.7367,B 24.9417,C -1.7633,E1 25.0402,E2 165.21} C_DIS
LIN {X 26.9255,Y -97.1779,Z 98,A -78.3552,B 24.9412,C -1.7711,E1 25.0439,E2 163.8125} C_DIS
Enddeposition()
END
